LIN {X 0,Y 170.14,Z 485.3,A -85,B 0,C 180,E1 -24974.606,E2 -24974.606} C_VEL
LIN {X 0,Y 177.602,Z 482.481,A -85,B 0,C 180,E1 -24977.722,E2 -24977.722} C_VEL
LIN {X 0,Y 183.018,Z 480.013,A -85,B 0,C 180,E1 -24980.176,E2 -24980.176} C_VEL
LIN {X 0,Y 180.641,Z 479.716,A -85,B 0,C 180,E1 -24981.501,E2 -24981.501} C_VEL
LIN {X 0,Y 171.109,Z 479.234,A -85,B 0,C 180,E1 -24984.898,E2 -24984.898} C_VEL
LIN {X 0,Y 162.459,Z 477.57,A -85,B 0,C 180,E1 -24988.726,E2 -24988.726} C_VEL
LIN {X 0,Y 154.788,Z 474.682,A -85,B 0,C 180,E1 -24992.996,E2 -24992.996} C_VEL
LIN {X 0,Y 148.331,Z 470.573,A -85,B 0,C 180,E1 -24997.725,E2 -24997.725} C_VEL
LIN {X 0,Y 146.154,Z 468.596,A -85,B 0,C 180,E1 -24999.725,E2 -24999.725} C_VEL
LIN {X 0,Y 143.595,Z 466.459,A -85,B 0,C 180,E1 -25001.638,E2 -25001.638} C_VEL
LIN {X 0,Y 138.227,Z 462.461,A -85,B 0,C 180,E1 -25004.589,E2 -25004.589} C_VEL
LIN {X 0,Y 133.314,Z 457.777,A -85,B 0,C 180,E1 -25007.666,E2 -25007.666} C_VEL
LIN {X 0,Y 131.549,Z 454.712,A -85,B 0,C 180,E1 -25009.741,E2 -25009.741} C_VEL
LIN {X 0,Y 129.832,Z 446.19,A -85,B 0,C 180,E1 -25015.342,E2 -25015.342} C_VEL
LIN {X 0,Y 129.143,Z 437.874,A -85,B 0,C 180,E1 -25019.999,E2 -25019.999} C_VEL
LIN {X 0,Y 129.267,Z 426.337,A -85,B 0,C 180,E1 -25025.459,E2 -25025.459} C_VEL
LIN {X 0,Y 130.008,Z 415.476,A -85,B 0,C 180,E1 -25029.725,E2 -25029.725} C_VEL
LIN {X 0,Y 131.217,Z 402.421,A -85,B 0,C 180,E1 -25033.911,E2 -25033.911} C_VEL
LIN {X 0,Y 132.163,Z 391.334,A -85,B 0,C 180,E1 -25036.826,E2 -25036.826} C_VEL
LIN {X 0,Y 129.638,Z 379.334,A -85,B 0,C 180,E1 -25039.29,E2 -25039.29} C_VEL
LIN {X 0,Y 129.065,Z 379.401,A -85,B 0,C 180,E1 -25045.825,E2 -25045.825} C_VEL
LIN {X 0,Y 129.036,Z 379.412,A -85,B 0,C 180,E1 -25049.373,E2 -25049.373} C_VEL
LIN {X 0,Y 128.998,Z 379.412,A -85,B 0,C 180,E1 -25055.192,E2 -25055.192} C_VEL
LIN {X 0,Y 128.993,Z 379.414,A -85,B 0,C 180,E1 -25060.828,E2 -25060.828} C_VEL
LIN {X 0,Y 128.966,Z 379.42,A -85,B 0,C 180,E1 -25065.107,E2 -25065.107} C_VEL
LIN {X 0,Y 128.959,Z 379.418,A -85,B 0,C 180,E1 -25069.726,E2 -25069.726} C_VEL
LIN {X 0,Y 128.993,Z 379.418,A -85,B 0,C 180,E1 -25074.81,E2 -25074.81} C_VEL
LIN {X 0,Y 129.033,Z 379.406,A -85,B 0,C 180,E1 -25080.646,E2 -25080.646} C_VEL
LIN {X 0,Y 129.136,Z 379.395,A -85,B 0,C 180,E1 -25087.607,E2 -25087.607} C_VEL
LIN {X 0,Y 129.18,Z 379.392,A -85,B 0,C 180,E1 -25090.948,E2 -25090.948} C_VEL
LIN {X 0,Y 129.367,Z 379.364,A -85,B 0,C 180,E1 -25097.921,E2 -25097.921} C_VEL
LIN {X 0,Y 129.477,Z 379.357,A -85,B 0,C 180,E1 -25100.628,E2 -25100.628} C_VEL
LIN {X 0,Y 130.089,Z 379.282,A -85,B 0,C 180,E1 -25110,E2 -25110} C_VEL
LIN {X 0,Y 129.478,Z 379.357,A -85,B 0,C 180,E1 -25119.372,E2 -25119.372} C_VEL
LIN {X 0,Y 129.345,Z 379.366,A -85,B 0,C 180,E1 -25122.553,E2 -25122.553} C_VEL
LIN {X 0,Y 129.158,Z 379.395,A -85,B 0,C 180,E1 -25129.056,E2 -25129.056} C_VEL
LIN {X 0,Y 129.109,Z 379.398,A -85,B 0,C 180,E1 -25132.399,E2 -25132.399} C_VEL
LIN {X 0,Y 129.036,Z 379.406,A -85,B 0,C 180,E1 -25139.374,E2 -25139.374} C_VEL
LIN {X 0,Y 129.026,Z 379.414,A -85,B 0,C 180,E1 -25145.21,E2 -25145.21} C_VEL
LIN {X 0,Y 129.007,Z 379.413,A -85,B 0,C 180,E1 -25150.824,E2 -25150.824} C_VEL
LIN {X 0,Y 128.972,Z 379.417,A -85,B 0,C 180,E1 -25155.106,E2 -25155.106} C_VEL
LIN {X 0,Y 128.955,Z 379.421,A -85,B 0,C 180,E1 -25159.73,E2 -25159.73} C_VEL
LIN {X 0,Y 128.963,Z 379.416,A -85,B 0,C 180,E1 -25164.831,E2 -25164.831} C_VEL
LIN {X 0,Y 129.052,Z 379.41,A -85,B 0,C 180,E1 -25170.652,E2 -25170.652} C_VEL
LIN {X 0,Y 129.11,Z 379.402,A -85,B 0,C 180,E1 -25177.728,E2 -25177.728} C_VEL
LIN {X 0,Y 129.166,Z 379.392,A -85,B 0,C 180,E1 -25180.946,E2 -25180.946} C_VEL
LIN {X 0,Y 129.421,Z 379.363,A -85,B 0,C 180,E1 -25187.815,E2 -25187.815} C_VEL
LIN {X 0,Y 129.534,Z 379.344,A -85,B 0,C 180,E1 -25190.633,E2 -25190.633} C_VEL
LIN {X 0,Y 130.092,Z 379.274,A -85,B 0,C 180,E1 -25200,E2 -25200} C_VEL
LIN {X 0,Y 129.48,Z 379.351,A -85,B 0,C 180,E1 -25209.372,E2 -25209.372} C_VEL
LIN {X 0,Y 129.347,Z 379.373,A -85,B 0,C 180,E1 -25212.553,E2 -25212.553} C_VEL
LIN {X 0,Y 129.157,Z 379.394,A -85,B 0,C 180,E1 -25219.056,E2 -25219.056} C_VEL
LIN {X 0,Y 129.111,Z 379.402,A -85,B 0,C 180,E1 -25222.398,E2 -25222.398} C_VEL
LIN {X 0,Y 129.038,Z 379.411,A -85,B 0,C 180,E1 -25229.373,E2 -25229.373} C_VEL
LIN {X 0,Y 129.053,Z 379.404,A -85,B 0,C 180,E1 -25235.226,E2 -25235.226} C_VEL
LIN {X 0,Y 129.361,Z 379.369,A -85,B 0,C 180,E1 -25240.689,E2 -25240.689} C_VEL
LIN {X 0,Y 129.959,Z 379.326,A -85,B 0,C 180,E1 -25245.132,E2 -25245.132} C_VEL
LIN {X 0,Y 131.308,Z 383.898,A -85,B 0,C 180,E1 -25250.037,E2 -25250.037} C_VEL
LIN {X 0,Y 131.527,Z 385.753,A -85,B 0,C 180,E1 -25252.017,E2 -25252.017} C_VEL
LIN {X 0,Y 130.174,Z 390.538,A -85,B 0,C 180,E1 -25257.323,E2 -25257.323} C_VEL
LIN {X 0,Y 128.998,Z 398.088,A -85,B 0,C 180,E1 -25265.989,E2 -25265.989} C_VEL
LIN {X 0,Y 128.362,Z 411.728,A -85,B 0,C 180,E1 -25268.252,E2 -25268.252} C_VEL
LIN {X 0,Y 128.633,Z 424.364,A -85,B 0,C 180,E1 -25270.863,E2 -25270.863} C_VEL
LIN {X 0,Y 129.819,Z 437.824,A -85,B 0,C 180,E1 -25274.295,E2 -25274.295} C_VEL
LIN {X 0,Y 131.612,Z 449.97,A -85,B 0,C 180,E1 -25278.058,E2 -25278.058} C_VEL
LIN {X 0,Y 132.698,Z 455.665,A -85,B 0,C 180,E1 -25280.088,E2 -25280.088} C_VEL
LIN {X 0,Y 133.201,Z 464.15,A -85,B 0,C 180,E1 -25283.942,E2 -25283.942} C_VEL
LIN {X 0,Y 133.939,Z 470.787,A -85,B 0,C 180,E1 -25287.567,E2 -25287.567} C_VEL
LIN {X 0,Y 135.046,Z 476.747,A -85,B 0,C 180,E1 -25291.491,E2 -25291.491} C_VEL
LIN {X 0,Y 134.77,Z 478.314,A -85,B 0,C 180,E1 -25292.989,E2 -25292.989} C_VEL
LIN {X 0,Y 132.305,Z 482.493,A -85,B 0,C 180,E1 -25299.17,E2 -25299.17} C_VEL
LIN {X 0,Y 131.65,Z 485.641,A -85,B 0,C 180,E1 -25306.071,E2 -25306.071} C_VEL
LIN {X 0,Y 132.923,Z 487.379,A -85,B 0,C 180,E1 -25311.722,E2 -25311.722} C_VEL
LIN {X 0,Y 136.259,Z 488.459,A -85,B 0,C 180,E1 -25317.659,E2 -25317.659} C_VEL
LIN {X 0,Y 141.551,Z 488.732,A -85,B 0,C 180,E1 -25323.103,E2 -25323.103} C_VEL
LIN {X 0,Y 148.341,Z 488.17,A -85,B 0,C 180,E1 -25328.018,E2 -25328.018} C_VEL
LIN {X 0,Y 156.192,Z 486.763,A -85,B 0,C 180,E1 -25332.45,E2 -25332.45} C_VEL
LIN {X 0,Y 165.142,Z 484.583,A -85,B 0,C 180,E1 -25336.342,E2 -25336.342} C_VEL
LIN {X 0,Y 172.211,Z 482.323,A -85,B 0,C 180,E1 -25339.234,E2 -25339.234} C_VEL
LIN {X 0,Y 174.086,Z 481.574,A -85,B 0,C 180,E1 -25340.09,E2 -25340.09} C_VEL
LIN {X 0,Y 169.266,Z 480.977,A -85,B 0,C 180,E1 -25342.082,E2 -25342.082} C_VEL
LIN {X 0,Y 160.81,Z 479.531,A -85,B 0,C 180,E1 -25345.378,E2 -25345.378} C_VEL
LIN {X 0,Y 152.361,Z 476.82,A -85,B 0,C 180,E1 -25349.509,E2 -25349.509} C_VEL
LIN {X 0,Y 144.959,Z 472.908,A -85,B 0,C 180,E1 -25354.129,E2 -25354.129} C_VEL
LIN {X 0,Y 138.954,Z 467.741,A -85,B 0,C 180,E1 -25359.265,E2 -25359.265} C_VEL
LIN {X 0,Y 134.271,Z 461.25,A -85,B 0,C 180,E1 -25364.828,E2 -25364.828} C_VEL
LIN {X 0,Y 131.549,Z 454.712,A -85,B 0,C 180,E1 -25369.741,E2 -25369.741} C_VEL
LIN {X 0,Y 130.004,Z 451.514,A -85,B 0,C 180,E1 -25371.813,E2 -25371.813} C_VEL
LIN {X 0,Y 126.277,Z 445.65,A -85,B 0,C 180,E1 -25374.992,E2 -25374.992} C_VEL
LIN {X 0,Y 122.987,Z 439.301,A -85,B 0,C 180,E1 -25378.18,E2 -25378.18} C_VEL
LIN {X 0,Y 122.189,Z 435.308,A -85,B 0,C 180,E1 -25380.201,E2 -25380.201} C_VEL
LIN {X 0,Y 122.392,Z 423.535,A -85,B 0,C 180,E1 -25385.767,E2 -25385.767} C_VEL
LIN {X 0,Y 123.115,Z 413.168,A -85,B 0,C 180,E1 -25389.86,E2 -25389.86} C_VEL
LIN {X 0,Y 124.272,Z 400.77,A -85,B 0,C 180,E1 -25393.907,E2 -25393.907} C_VEL
LIN {X 0,Y 125.093,Z 391.958,A -85,B 0,C 180,E1 -25396.314,E2 -25396.314} C_VEL
LIN {X 0,Y 122.644,Z 380.202,A -85,B 0,C 180,E1 -25398.911,E2 -25398.911} C_VEL
LIN {X 0,Y 121.974,Z 380.289,A -85,B 0,C 180,E1 -25407.448,E2 -25407.448} C_VEL
LIN {X 0,Y 121.913,Z 380.298,A -85,B 0,C 180,E1 -25411.253,E2 -25411.253} C_VEL
LIN {X 0,Y 121.922,Z 380.294,A -85,B 0,C 180,E1 -25416.195,E2 -25416.195} C_VEL
LIN {X 0,Y 121.92,Z 380.293,A -85,B 0,C 180,E1 -25421.464,E2 -25421.464} C_VEL
LIN {X 0,Y 121.891,Z 380.301,A -85,B 0,C 180,E1 -25428.551,E2 -25428.551} C_VEL
LIN {X 0,Y 121.946,Z 380.296,A -85,B 0,C 180,E1 -25434.808,E2 -25434.808} C_VEL
LIN {X 0,Y 121.942,Z 380.289,A -85,B 0,C 180,E1 -25439.826,E2 -25439.826} C_VEL
LIN {X 0,Y 122.068,Z 380.275,A -85,B 0,C 180,E1 -25447.1,E2 -25447.1} C_VEL
LIN {X 0,Y 122.122,Z 380.272,A -85,B 0,C 180,E1 -25453.277,E2 -25453.277} C_VEL
LIN {X 0,Y 122.318,Z 380.241,A -85,B 0,C 180,E1 -25457.623,E2 -25457.623} C_VEL
LIN {X 0,Y 122.426,Z 380.233,A -85,B 0,C 180,E1 -25463.407,E2 -25463.407} C_VEL
LIN {X 0,Y 123.043,Z 380.159,A -85,B 0,C 180,E1 -25470,E2 -25470} C_VEL
LIN {X 0,Y 122.427,Z 380.233,A -85,B 0,C 180,E1 -25476.593,E2 -25476.593} C_VEL
LIN {X 0,Y 122.318,Z 380.241,A -85,B 0,C 180,E1 -25482.377,E2 -25482.377} C_VEL
LIN {X 0,Y 122.112,Z 380.273,A -85,B 0,C 180,E1 -25486.725,E2 -25486.725} C_VEL
LIN {X 0,Y 122.024,Z 380.281,A -85,B 0,C 180,E1 -25492.852,E2 -25492.852} C_VEL
LIN {X 0,Y 121.95,Z 380.293,A -85,B 0,C 180,E1 -25497.455,E2 -25497.455} C_VEL
LIN {X 0,Y 121.913,Z 380.294,A -85,B 0,C 180,E1 -25501.254,E2 -25501.254} C_VEL
LIN {X 0,Y 121.939,Z 380.293,A -85,B 0,C 180,E1 -25506.207,E2 -25506.207} C_VEL
LIN {X 0,Y 121.931,Z 380.296,A -85,B 0,C 180,E1 -25511.47,E2 -25511.47} C_VEL
LIN {X 0,Y 121.892,Z 380.297,A -85,B 0,C 180,E1 -25518.552,E2 -25518.552} C_VEL
LIN {X 0,Y 121.915,Z 380.293,A -85,B 0,C 180,E1 -25524.798,E2 -25524.798} C_VEL
LIN {X 0,Y 121.941,Z 380.295,A -85,B 0,C 180,E1 -25529.829,E2 -25529.829} C_VEL
LIN {X 0,Y 121.986,Z 380.287,A -85,B 0,C 180,E1 -25536.216,E2 -25536.216} C_VEL
LIN {X 0,Y 122.054,Z 380.28,A -85,B 0,C 180,E1 -25539.789,E2 -25539.789} C_VEL
LIN {X 0,Y 122.289,Z 380.253,A -85,B 0,C 180,E1 -25546.71,E2 -25546.71} C_VEL
LIN {X 0,Y 122.46,Z 380.228,A -85,B 0,C 180,E1 -25550.086,E2 -25550.086} C_VEL
LIN {X 0,Y 122.614,Z 380.211,A -85,B 0,C 180,E1 -25556.715,E2 -25556.715} C_VEL
LIN {X 0,Y 123.045,Z 380.151,A -85,B 0,C 180,E1 -25560.001,E2 -25560.001} C_VEL
LIN {X 0,Y 122.428,Z 380.232,A -85,B 0,C 180,E1 -25566.593,E2 -25566.593} C_VEL
LIN {X 0,Y 122.32,Z 380.249,A -85,B 0,C 180,E1 -25572.377,E2 -25572.377} C_VEL
LIN {X 0,Y 122.111,Z 380.267,A -85,B 0,C 180,E1 -25576.725,E2 -25576.725} C_VEL
LIN {X 0,Y 122.026,Z 380.283,A -85,B 0,C 180,E1 -25582.851,E2 -25582.851} C_VEL
LIN {X 0,Y 121.952,Z 380.29,A -85,B 0,C 180,E1 -25587.454,E2 -25587.454} C_VEL
LIN {X 0,Y 121.917,Z 380.298,A -85,B 0,C 180,E1 -25591.253,E2 -25591.253} C_VEL
LIN {X 0,Y 122.037,Z 380.282,A -85,B 0,C 180,E1 -25596.268,E2 -25596.268} C_VEL
LIN {X 0,Y 122.898,Z 380.18,A -85,B 0,C 180,E1 -25605.125,E2 -25605.125} C_VEL
LIN {X 0,Y 123.1,Z 380.269,A -85,B 0,C 180,E1 -25606.284,E2 -25606.284} C_VEL
LIN {X 0,Y 124.019,Z 383.15,A -85,B 0,C 180,E1 -25609.562,E2 -25609.562} C_VEL
LIN {X 0,Y 124.38,Z 385.558,A -85,B 0,C 180,E1 -25612.286,E2 -25612.286} C_VEL
LIN {X 0,Y 123.156,Z 389.67,A -85,B 0,C 180,E1 -25617.171,E2 -25617.171} C_VEL
LIN {X 0,Y 122.005,Z 397.074,A -85,B 0,C 180,E1 -25626.298,E2 -25626.298} C_VEL
LIN {X 0,Y 121.409,Z 409.093,A -85,B 0,C 180,E1 -25628.377,E2 -25628.377} C_VEL
LIN {X 0,Y 121.725,Z 423.36,A -85,B 0,C 180,E1 -25631.485,E2 -25631.485} C_VEL
LIN {X 0,Y 123.055,Z 437.085,A -85,B 0,C 180,E1 -25635.204,E2 -25635.204} C_VEL
LIN {X 0,Y 124.946,Z 448.82,A -85,B 0,C 180,E1 -25639.056,E2 -25639.056} C_VEL
LIN {X 0,Y 126.146,Z 454.516,A -85,B 0,C 180,E1 -25641.187,E2 -25641.187} C_VEL
LIN {X 0,Y 126.68,Z 461.745,A -85,B 0,C 180,E1 -25644.633,E2 -25644.633} C_VEL
LIN {X 0,Y 127.616,Z 468.962,A -85,B 0,C 180,E1 -25648.725,E2 -25648.725} C_VEL
LIN {X 0,Y 128.474,Z 473.274,A -85,B 0,C 180,E1 -25651.567,E2 -25651.567} C_VEL
LIN {X 0,Y 128.453,Z 475.044,A -85,B 0,C 180,E1 -25653.136,E2 -25653.136} C_VEL
LIN {X 0,Y 125.905,Z 479.435,A -85,B 0,C 180,E1 -25659.64,E2 -25659.64} C_VEL
LIN {X 0,Y 125.383,Z 483.15,A -85,B 0,C 180,E1 -25667.655,E2 -25667.655} C_VEL
LIN {X 0,Y 128.252,Z 485.578,A -85,B 0,C 180,E1 -25676.001,E2 -25676.001} C_VEL
LIN {X 0,Y 133.627,Z 486.621,A -85,B 0,C 180,E1 -25682.699,E2 -25682.699} C_VEL
LIN {X 0,Y 142.919,Z 486.504,A -85,B 0,C 180,E1 -25689.738,E2 -25689.738} C_VEL
LIN {X 0,Y 151.093,Z 485.444,A -85,B 0,C 180,E1 -25694.244,E2 -25694.244} C_VEL
LIN {X 0,Y 160.329,Z 483.66,A -85,B 0,C 180,E1 -25698.176,E2 -25698.176} C_VEL
LIN {X 0,Y 165.008,Z 482.426,A -85,B 0,C 180,E1 -25700.054,E2 -25700.054} C_VEL
LIN {X 0,Y 159.837,Z 481.469,A -85,B 0,C 180,E1 -25702.006,E2 -25702.006} C_VEL
LIN {X 0,Y 150.542,Z 478.882,A -85,B 0,C 180,E1 -25705.929,E2 -25705.929} C_VEL
LIN {X 0,Y 142.294,Z 475.138,A -85,B 0,C 180,E1 -25710.402,E2 -25710.402} C_VEL
LIN {X 0,Y 135.297,Z 470.197,A -85,B 0,C 180,E1 -25715.445,E2 -25715.445} C_VEL
LIN {X 0,Y 129.736,Z 463.945,A -85,B 0,C 180,E1 -25721.032,E2 -25721.032} C_VEL
LIN {X 0,Y 125.658,Z 456.29,A -85,B 0,C 180,E1 -25727.072,E2 -25727.072} C_VEL
LIN {X 0,Y 123.222,Z 447.02,A -85,B 0,C 180,E1 -25733.449,E2 -25733.449} C_VEL
LIN {X 0,Y 122.396,Z 438.754,A -85,B 0,C 180,E1 -25738.354,E2 -25738.354} C_VEL
LIN {X 0,Y 122.189,Z 435.308,A -85,B 0,C 180,E1 -25740.201,E2 -25740.201} C_VEL
LIN {X 0,Y 121.505,Z 431.227,A -85,B 0,C 180,E1 -25742.158,E2 -25742.158} C_VEL
LIN {X 0,Y 118.944,Z 423.968,A -85,B 0,C 180,E1 -25745.092,E2 -25745.092} C_VEL
LIN {X 0,Y 116.555,Z 416.203,A -85,B 0,C 180,E1 -25747.953,E2 -25747.953} C_VEL
LIN {X 0,Y 116.228,Z 411.378,A -85,B 0,C 180,E1 -25749.71,E2 -25749.71} C_VEL
LIN {X 0,Y 117.336,Z 399.012,A -85,B 0,C 180,E1 -25753.862,E2 -25753.862} C_VEL
LIN {X 0,Y 117.981,Z 391.979,A -85,B 0,C 180,E1 -25755.837,E2 -25755.837} C_VEL
LIN {X 0,Y 115.703,Z 381.064,A -85,B 0,C 180,E1 -25758.366,E2 -25758.366} C_VEL
LIN {X 0,Y 114.949,Z 381.159,A -85,B 0,C 180,E1 -25765.339,E2 -25765.339} C_VEL
LIN {X 0,Y 114.871,Z 381.176,A -85,B 0,C 180,E1 -25771.069,E2 -25771.069} C_VEL
LIN {X 0,Y 114.822,Z 381.182,A -85,B 0,C 180,E1 -25777.739,E2 -25777.739} C_VEL
LIN {X 0,Y 114.832,Z 381.174,A -85,B 0,C 180,E1 -25782.741,E2 -25782.741} C_VEL
LIN {X 0,Y 114.819,Z 381.182,A -85,B 0,C 180,E1 -25787.677,E2 -25787.677} C_VEL
LIN {X 0,Y 114.812,Z 381.178,A -85,B 0,C 180,E1 -25792.727,E2 -25792.727} C_VEL
LIN {X 0,Y 114.869,Z 381.17,A -85,B 0,C 180,E1 -25798.931,E2 -25798.931} C_VEL
LIN {X 0,Y 114.966,Z 381.161,A -85,B 0,C 180,E1 -25806.485,E2 -25806.485} C_VEL
LIN {X 0,Y 115.027,Z 381.157,A -85,B 0,C 180,E1 -25812.212,E2 -25812.212} C_VEL
LIN {X 0,Y 115.252,Z 381.121,A -85,B 0,C 180,E1 -25817.333,E2 -25817.333} C_VEL
LIN {X 0,Y 115.367,Z 381.113,A -85,B 0,C 180,E1 -25823.002,E2 -25823.002} C_VEL
LIN {X 0,Y 115.994,Z 381.037,A -85,B 0,C 180,E1 -25830,E2 -25830} C_VEL
LIN {X 0,Y 115.367,Z 381.113,A -85,B 0,C 180,E1 -25836.998,E2 -25836.998} C_VEL
LIN {X 0,Y 115.252,Z 381.121,A -85,B 0,C 180,E1 -25842.667,E2 -25842.667} C_VEL
LIN {X 0,Y 115.014,Z 381.159,A -85,B 0,C 180,E1 -25847.79,E2 -25847.79} C_VEL
LIN {X 0,Y 114.947,Z 381.164,A -85,B 0,C 180,E1 -25853.493,E2 -25853.493} C_VEL
LIN {X 0,Y 114.87,Z 381.17,A -85,B 0,C 180,E1 -25861.069,E2 -25861.069} C_VEL
LIN {X 0,Y 114.849,Z 381.172,A -85,B 0,C 180,E1 -25867.73,E2 -25867.73} C_VEL
LIN {X 0,Y 114.842,Z 381.18,A -85,B 0,C 180,E1 -25872.747,E2 -25872.747} C_VEL
LIN {X 0,Y 114.821,Z 381.176,A -85,B 0,C 180,E1 -25877.679,E2 -25877.679} C_VEL
LIN {X 0,Y 114.795,Z 381.186,A -85,B 0,C 180,E1 -25882.74,E2 -25882.74} C_VEL
LIN {X 0,Y 114.864,Z 381.177,A -85,B 0,C 180,E1 -25888.938,E2 -25888.938} C_VEL
LIN {X 0,Y 114.949,Z 381.164,A -85,B 0,C 180,E1 -25896.508,E2 -25896.508} C_VEL
LIN {X 0,Y 115.023,Z 381.151,A -85,B 0,C 180,E1 -25902.212,E2 -25902.212} C_VEL
LIN {X 0,Y 115.289,Z 381.124,A -85,B 0,C 180,E1 -25907.258,E2 -25907.258} C_VEL
LIN {X 0,Y 115.396,Z 381.108,A -85,B 0,C 180,E1 -25909.473,E2 -25909.473} C_VEL
LIN {X 0,Y 115.541,Z 381.093,A -85,B 0,C 180,E1 -25916.513,E2 -25916.513} C_VEL
LIN {X 0,Y 115.997,Z 381.029,A -85,B 0,C 180,E1 -25920.001,E2 -25920.001} C_VEL
LIN {X 0,Y 115.369,Z 381.11,A -85,B 0,C 180,E1 -25926.999,E2 -25926.999} C_VEL
LIN {X 0,Y 115.255,Z 381.129,A -85,B 0,C 180,E1 -25932.667,E2 -25932.667} C_VEL
LIN {X 0,Y 115.014,Z 381.151,A -85,B 0,C 180,E1 -25937.791,E2 -25937.791} C_VEL
LIN {X 0,Y 114.95,Z 381.165,A -85,B 0,C 180,E1 -25943.493,E2 -25943.493} C_VEL
LIN {X 0,Y 114.874,Z 381.175,A -85,B 0,C 180,E1 -25951.07,E2 -25951.07} C_VEL
LIN {X 0,Y 115.033,Z 381.155,A -85,B 0,C 180,E1 -25957.659,E2 -25957.659} C_VEL
LIN {X 0,Y 116.078,Z 381.03,A -85,B 0,C 180,E1 -25966.599,E2 -25966.599} C_VEL
LIN {X 0,Y 116.265,Z 381.092,A -85,B 0,C 180,E1 -25967.535,E2 -25967.535} C_VEL
LIN {X 0,Y 117.185,Z 384.161,A -85,B 0,C 180,E1 -25971.23,E2 -25971.23} C_VEL
LIN {X 0,Y 117.073,Z 385.702,A -85,B 0,C 180,E1 -25973.107,E2 -25973.107} C_VEL
LIN {X 0,Y 115.477,Z 391.71,A -85,B 0,C 180,E1 -25980.863,E2 -25980.863} C_VEL
LIN {X 0,Y 115.018,Z 396.094,A -85,B 0,C 180,E1 -25986.675,E2 -25986.675} C_VEL
LIN {X 0,Y 114.46,Z 407.836,A -85,B 0,C 180,E1 -25988.854,E2 -25988.854} C_VEL
LIN {X 0,Y 114.832,Z 422.144,A -85,B 0,C 180,E1 -25992.18,E2 -25992.18} C_VEL
LIN {X 0,Y 116.245,Z 435.48,A -85,B 0,C 180,E1 -25996.005,E2 -25996.005} C_VEL
LIN {X 0,Y 118.355,Z 447.553,A -85,B 0,C 180,E1 -26000.17,E2 -26000.17} C_VEL
LIN {X 0,Y 119.663,Z 453.235,A -85,B 0,C 180,E1 -26002.406,E2 -26002.406} C_VEL
LIN {X 0,Y 120.475,Z 461.551,A -85,B 0,C 180,E1 -26006.655,E2 -26006.655} C_VEL
LIN {X 0,Y 121.894,Z 469.512,A -85,B 0,C 180,E1 -26011.652,E2 -26011.652} C_VEL
LIN {X 0,Y 122.132,Z 471.597,A -85,B 0,C 180,E1 -26013.299,E2 -26013.299} C_VEL
LIN {X 0,Y 120.461,Z 474.552,A -85,B 0,C 180,E1 -26017.326,E2 -26017.326} C_VEL
LIN {X 0,Y 119.036,Z 478.093,A -85,B 0,C 180,E1 -26023.66,E2 -26023.66} C_VEL
LIN {X 0,Y 119.56,Z 480.975,A -85,B 0,C 180,E1 -26030.652,E2 -26030.652} C_VEL
LIN {X 0,Y 122.273,Z 482.983,A -85,B 0,C 180,E1 -26037.376,E2 -26037.376} C_VEL
LIN {X 0,Y 128.681,Z 484.429,A -85,B 0,C 180,E1 -26044.99,E2 -26044.99} C_VEL
LIN {X 0,Y 137.686,Z 484.661,A -85,B 0,C 180,E1 -26051.573,E2 -26051.573} C_VEL
LIN {X 0,Y 146.172,Z 483.928,A -85,B 0,C 180,E1 -26056.154,E2 -26056.154} C_VEL
LIN {X 0,Y 150.86,Z 483.324,A -85,B 0,C 180,E1 -26058.192,E2 -26058.192} C_VEL
LIN {X 0,Y 154.336,Z 482.295,A -85,B 0,C 180,E1 -26060.393,E2 -26060.393} C_VEL
LIN {X 0,Y 144.732,Z 479.243,A -85,B 0,C 180,E1 -26064.358,E2 -26064.358} C_VEL
LIN {X 0,Y 136.178,Z 475.05,A -85,B 0,C 180,E1 -26068.929,E2 -26068.929} C_VEL
LIN {X 0,Y 128.883,Z 469.671,A -85,B 0,C 180,E1 -26074.135,E2 -26074.135} C_VEL
LIN {X 0,Y 123.086,Z 463.014,A -85,B 0,C 180,E1 -26079.965,E2 -26079.965} C_VEL
LIN {X 0,Y 118.441,Z 453.782,A -85,B 0,C 180,E1 -26087.143,E2 -26087.143} C_VEL
LIN {X 0,Y 116.367,Z 445.166,A -85,B 0,C 180,E1 -26093.062,E2 -26093.062} C_VEL
LIN {X 0,Y 115.471,Z 436.462,A -85,B 0,C 180,E1 -26098.256,E2 -26098.256} C_VEL
LIN {X 0,Y 115.407,Z 424.357,A -85,B 0,C 180,E1 -26104.365,E2 -26104.365} C_VEL
LIN {X 0,Y 116.038,Z 414.064,A -85,B 0,C 180,E1 -26108.708,E2 -26108.708} C_VEL
LIN {X 0,Y 116.228,Z 411.378,A -85,B 0,C 180,E1 -26109.71,E2 -26109.71} C_VEL
LIN {X 0,Y 115.939,Z 406.526,A -85,B 0,C 180,E1 -26111.367,E2 -26111.367} C_VEL
LIN {X 0,Y 114.723,Z 401.509,A -85,B 0,C 180,E1 -26112.857,E2 -26112.857} C_VEL
LIN {X 0,Y 111.131,Z 391.201,A -85,B 0,C 180,E1 -26115.515,E2 -26115.515} C_VEL
LIN {X 0,Y 109.189,Z 384.008,A -85,B 0,C 180,E1 -26117.164,E2 -26117.164} C_VEL
LIN {X 0,Y 108.789,Z 381.923,A -85,B 0,C 180,E1 -26117.674,E2 -26117.674} C_VEL
LIN {X 0,Y 107.83,Z 382.048,A -85,B 0,C 180,E1 -26127.144,E2 -26127.144} C_VEL
LIN {X 0,Y 107.797,Z 382.055,A -85,B 0,C 180,E1 -26132.053,E2 -26132.053} C_VEL
LIN {X 0,Y 107.729,Z 382.066,A -85,B 0,C 180,E1 -26138.477,E2 -26138.477} C_VEL
LIN {X 0,Y 107.705,Z 382.068,A -85,B 0,C 180,E1 -26145.87,E2 -26145.87} C_VEL
LIN {X 0,Y 107.71,Z 382.06,A -85,B 0,C 180,E1 -26151.534,E2 -26151.534} C_VEL
LIN {X 0,Y 107.807,Z 382.051,A -85,B 0,C 180,E1 -26158.566,E2 -26158.566} C_VEL
LIN {X 0,Y 107.931,Z 382.036,A -85,B 0,C 180,E1 -26167.002,E2 -26167.002} C_VEL
LIN {X 0,Y 108.036,Z 382.025,A -85,B 0,C 180,E1 -26174.918,E2 -26174.918} C_VEL
LIN {X 0,Y 108.254,Z 381.997,A -85,B 0,C 180,E1 -26178.769,E2 -26178.769} C_VEL
LIN {X 0,Y 108.448,Z 381.97,A -85,B 0,C 180,E1 -26186.285,E2 -26186.285} C_VEL
LIN {X 0,Y 108.944,Z 381.915,A -85,B 0,C 180,E1 -26190,E2 -26190} C_VEL
LIN {X 0,Y 108.305,Z 381.993,A -85,B 0,C 180,E1 -26197.457,E2 -26197.457} C_VEL
LIN {X 0,Y 108.173,Z 382.002,A -85,B 0,C 180,E1 -26202.957,E2 -26202.957} C_VEL
LIN {X 0,Y 107.906,Z 382.042,A -85,B 0,C 180,E1 -26209.006,E2 -26209.006} C_VEL
LIN {X 0,Y 107.858,Z 382.049,A -85,B 0,C 180,E1 -26214.185,E2 -26214.185} C_VEL
LIN {X 0,Y 107.8,Z 382.055,A -85,B 0,C 180,E1 -26222.057,E2 -26222.057} C_VEL
LIN {X 0,Y 107.751,Z 382.055,A -85,B 0,C 180,E1 -26228.493,E2 -26228.493} C_VEL
LIN {X 0,Y 107.709,Z 382.063,A -85,B 0,C 180,E1 -26235.87,E2 -26235.87} C_VEL
LIN {X 0,Y 107.699,Z 382.07,A -85,B 0,C 180,E1 -26241.544,E2 -26241.544} C_VEL
LIN {X 0,Y 107.799,Z 382.055,A -85,B 0,C 180,E1 -26248.564,E2 -26248.564} C_VEL
LIN {X 0,Y 107.913,Z 382.042,A -85,B 0,C 180,E1 -26256.999,E2 -26256.999} C_VEL
LIN {X 0,Y 108.049,Z 382.023,A -85,B 0,C 180,E1 -26264.92,E2 -26264.92} C_VEL
LIN {X 0,Y 108.309,Z 381.992,A -85,B 0,C 180,E1 -26268.775,E2 -26268.775} C_VEL
LIN {X 0,Y 108.466,Z 381.975,A -85,B 0,C 180,E1 -26276.286,E2 -26276.286} C_VEL
LIN {X 0,Y 108.946,Z 381.907,A -85,B 0,C 180,E1 -26280.001,E2 -26280.001} C_VEL
LIN {X 0,Y 108.307,Z 381.989,A -85,B 0,C 180,E1 -26287.457,E2 -26287.457} C_VEL
LIN {X 0,Y 108.175,Z 382.01,A -85,B 0,C 180,E1 -26292.956,E2 -26292.956} C_VEL
LIN {X 0,Y 107.907,Z 382.041,A -85,B 0,C 180,E1 -26299.006,E2 -26299.006} C_VEL
LIN {X 0,Y 107.86,Z 382.045,A -85,B 0,C 180,E1 -26304.185,E2 -26304.185} C_VEL
LIN {X 0,Y 107.808,Z 382.053,A -85,B 0,C 180,E1 -26312.061,E2 -26312.061} C_VEL
LIN {X 0,Y 108.147,Z 382.012,A -85,B 0,C 180,E1 -26320.532,E2 -26320.532} C_VEL
LIN {X 0,Y 109.512,Z 381.873,A -85,B 0,C 180,E1 -26328.944,E2 -26328.944} C_VEL
LIN {X 0,Y 109.851,Z 382.874,A -85,B 0,C 180,E1 -26330.224,E2 -26330.224} C_VEL
LIN {X 0,Y 110.024,Z 384.729,A -85,B 0,C 180,E1 -26332.639,E2 -26332.639} C_VEL
LIN {X 0,Y 108.724,Z 389.222,A -85,B 0,C 180,E1 -26338.86,E2 -26338.86} C_VEL
LIN {X 0,Y 108.067,Z 395.013,A -85,B 0,C 180,E1 -26347.159,E2 -26347.159} C_VEL
LIN {X 0,Y 107.551,Z 407.596,A -85,B 0,C 180,E1 -26349.687,E2 -26349.687} C_VEL
LIN {X 0,Y 107.99,Z 420.747,A -85,B 0,C 180,E1 -26352.97,E2 -26352.97} C_VEL
LIN {X 0,Y 109.543,Z 434.095,A -85,B 0,C 180,E1 -26357.027,E2 -26357.027} C_VEL
LIN {X 0,Y 111.83,Z 446.154,A -85,B 0,C 180,E1 -26361.416,E2 -26361.416} C_VEL
LIN {X 0,Y 113.366,Z 452.763,A -85,B 0,C 180,E1 -26364.214,E2 -26364.214} C_VEL
LIN {X 0,Y 114.508,Z 461.538,A -85,B 0,C 180,E1 -26369.121,E2 -26369.121} C_VEL
LIN {X 0,Y 115.894,Z 467.951,A -85,B 0,C 180,E1 -26373.476,E2 -26373.476} C_VEL
LIN {X 0,Y 114.516,Z 470.672,A -85,B 0,C 180,E1 -26377.05,E2 -26377.05} C_VEL
LIN {X 0,Y 112.839,Z 474.848,A -85,B 0,C 180,E1 -26384.426,E2 -26384.426} C_VEL
LIN {X 0,Y 113.477,Z 477.975,A -85,B 0,C 180,E1 -26391.814,E2 -26391.814} C_VEL
LIN {X 0,Y 116.446,Z 480.221,A -85,B 0,C 180,E1 -26398.871,E2 -26398.871} C_VEL
LIN {X 0,Y 121.651,Z 481.759,A -85,B 0,C 180,E1 -26405.29,E2 -26405.29} C_VEL
LIN {X 0,Y 128.602,Z 482.537,A -85,B 0,C 180,E1 -26410.98,E2 -26410.98} C_VEL
LIN {X 0,Y 141.463,Z 482.217,A -85,B 0,C 180,E1 -26418.178,E2 -26418.178} C_VEL
LIN {X 0,Y 144.373,Z 481.986,A -85,B 0,C 180,E1 -26419.436,E2 -26419.436} C_VEL
LIN {X 0,Y 143.839,Z 481.289,A -85,B 0,C 180,E1 -26420.566,E2 -26420.566} C_VEL
LIN {X 0,Y 134.455,Z 477.217,A -85,B 0,C 180,E1 -26424.902,E2 -26424.902} C_VEL
LIN {X 0,Y 126.146,Z 471.985,A -85,B 0,C 180,E1 -26429.905,E2 -26429.905} C_VEL
LIN {X 0,Y 119.372,Z 465.547,A -85,B 0,C 180,E1 -26435.661,E2 -26435.661} C_VEL
LIN {X 0,Y 114.101,Z 457.746,A -85,B 0,C 180,E1 -26442.062,E2 -26442.062} C_VEL
LIN {X 0,Y 110.576,Z 448.356,A -85,B 0,C 180,E1 -26449.007,E2 -26449.007} C_VEL
LIN {X 0,Y 109.025,Z 438.639,A -85,B 0,C 180,E1 -26455.378,E2 -26455.378} C_VEL
LIN {X 0,Y 108.438,Z 426.844,A -85,B 0,C 180,E1 -26461.856,E2 -26461.856} C_VEL
LIN {X 0,Y 109.015,Z 414.776,A -85,B 0,C 180,E1 -26467.408,E2 -26467.408} C_VEL
LIN {X 0,Y 110.104,Z 401.216,A -85,B 0,C 180,E1 -26472.44,E2 -26472.44} C_VEL
LIN {X 0,Y 110.894,Z 391.893,A -85,B 0,C 180,E1 -26475.275,E2 -26475.275} C_VEL
LIN {X 0,Y 109.189,Z 384.008,A -85,B 0,C 180,E1 -26477.164,E2 -26477.164} C_VEL
LIN {X 0,Y 108.623,Z 382.755,A -85,B 0,C 180,E1 -26477.814,E2 -26477.814} C_VEL
LIN {X 0,Y 107.486,Z 382.185,A -85,B 0,C 180,E1 -26479.145,E2 -26479.145} C_VEL
LIN {X 0,Y 104.036,Z 382.522,A -85,B 0,C 180,E1 -26483.899,E2 -26483.899} C_VEL
LIN {X 0,Y 101.665,Z 383.072,A -85,B 0,C 180,E1 -26488.763,E2 -26488.763} C_VEL
LIN {X 0,Y 100.686,Z 382.935,A -85,B 0,C 180,E1 -26493.879,E2 -26493.879} C_VEL
LIN {X 0,Y 100.678,Z 382.943,A -85,B 0,C 180,E1 -26499.836,E2 -26499.836} C_VEL
LIN {X 0,Y 100.676,Z 382.943,A -85,B 0,C 180,E1 -26505.726,E2 -26505.726} C_VEL
LIN {X 0,Y 100.649,Z 382.94,A -85,B 0,C 180,E1 -26511.065,E2 -26511.065} C_VEL
LIN {X 0,Y 100.7,Z 382.94,A -85,B 0,C 180,E1 -26516.876,E2 -26516.876} C_VEL
LIN {X 0,Y 100.786,Z 382.93,A -85,B 0,C 180,E1 -26525.267,E2 -26525.267} C_VEL
LIN {X 0,Y 100.835,Z 382.919,A -85,B 0,C 180,E1 -26529.605,E2 -26529.605} C_VEL
LIN {X 0,Y 101.102,Z 382.883,A -85,B 0,C 180,E1 -26536.702,E2 -26536.702} C_VEL
LIN {X 0,Y 101.243,Z 382.874,A -85,B 0,C 180,E1 -26542.02,E2 -26542.02} C_VEL
LIN {X 0,Y 101.867,Z 382.797,A -85,B 0,C 180,E1 -26550,E2 -26550} C_VEL
LIN {X 0,Y 101.244,Z 382.874,A -85,B 0,C 180,E1 -26557.981,E2 -26557.981} C_VEL
LIN {X 0,Y 101.102,Z 382.883,A -85,B 0,C 180,E1 -26563.299,E2 -26563.299} C_VEL
LIN {X 0,Y 100.817,Z 382.921,A -85,B 0,C 180,E1 -26570.399,E2 -26570.399} C_VEL
LIN {X 0,Y 100.774,Z 382.931,A -85,B 0,C 180,E1 -26574.959,E2 -26574.959} C_VEL
LIN {X 0,Y 100.708,Z 382.939,A -85,B 0,C 180,E1 -26583.131,E2 -26583.131} C_VEL
LIN {X 0,Y 100.694,Z 382.937,A -85,B 0,C 180,E1 -26589.849,E2 -26589.849} C_VEL
LIN {X 0,Y 100.68,Z 382.939,A -85,B 0,C 180,E1 -26595.73,E2 -26595.73} C_VEL
LIN {X 0,Y 100.64,Z 382.949,A -85,B 0,C 180,E1 -26601.061,E2 -26601.061} C_VEL
LIN {X 0,Y 100.693,Z 382.936,A -85,B 0,C 180,E1 -26606.884,E2 -26606.884} C_VEL
LIN {X 0,Y 100.787,Z 382.924,A -85,B 0,C 180,E1 -26615.268,E2 -26615.268} C_VEL
LIN {X 0,Y 100.822,Z 382.925,A -85,B 0,C 180,E1 -26619.603,E2 -26619.603} C_VEL
LIN {X 0,Y 101.202,Z 382.879,A -85,B 0,C 180,E1 -26627.976,E2 -26627.976} C_VEL
LIN {X 0,Y 101.282,Z 382.861,A -85,B 0,C 180,E1 -26632.023,E2 -26632.023} C_VEL
LIN {X 0,Y 101.87,Z 382.788,A -85,B 0,C 180,E1 -26640.001,E2 -26640.001} C_VEL
LIN {X 0,Y 101.246,Z 382.867,A -85,B 0,C 180,E1 -26647.981,E2 -26647.981} C_VEL
LIN {X 0,Y 101.104,Z 382.891,A -85,B 0,C 180,E1 -26653.299,E2 -26653.299} C_VEL
LIN {X 0,Y 100.818,Z 382.927,A -85,B 0,C 180,E1 -26660.399,E2 -26660.399} C_VEL
LIN {X 0,Y 100.777,Z 382.925,A -85,B 0,C 180,E1 -26664.959,E2 -26664.959} C_VEL
LIN {X 0,Y 100.752,Z 382.93,A -85,B 0,C 180,E1 -26673.167,E2 -26673.167} C_VEL
LIN {X 0,Y 101.056,Z 382.896,A -85,B 0,C 180,E1 -26680.092,E2 -26680.092} C_VEL
LIN {X 0,Y 102.427,Z 382.729,A -85,B 0,C 180,E1 -26689.006,E2 -26689.006} C_VEL
LIN {X 0,Y 102.805,Z 382.89,A -85,B 0,C 180,E1 -26690.977,E2 -26690.977} C_VEL
LIN {X 0,Y 102.673,Z 385.033,A -85,B 0,C 180,E1 -26694.048,E2 -26694.048} C_VEL
LIN {X 0,Y 101.114,Z 391.934,A -85,B 0,C 180,E1 -26704.634,E2 -26704.634} C_VEL
LIN {X 0,Y 101.143,Z 394.104,A -85,B 0,C 180,E1 -26707.8,E2 -26707.8} C_VEL
LIN {X 0,Y 100.693,Z 407.047,A -85,B 0,C 180,E1 -26710.638,E2 -26710.638} C_VEL
LIN {X 0,Y 101.329,Z 420.784,A -85,B 0,C 180,E1 -26714.365,E2 -26714.365} C_VEL
LIN {X 0,Y 103.125,Z 434.011,A -85,B 0,C 180,E1 -26718.7,E2 -26718.7} C_VEL
LIN {X 0,Y 105.714,Z 445.868,A -85,B 0,C 180,E1 -26723.337,E2 -26723.337} C_VEL
LIN {X 0,Y 107.067,Z 451.051,A -85,B 0,C 180,E1 -26725.661,E2 -26725.661} C_VEL
LIN {X 0,Y 108.2,Z 458.511,A -85,B 0,C 180,E1 -26730,E2 -26730} C_VEL
LIN {X 0,Y 109.403,Z 463.919,A -85,B 0,C 180,E1 -26733.683,E2 -26733.683} C_VEL
LIN {X 0,Y 109.199,Z 465.75,A -85,B 0,C 180,E1 -26735.54,E2 -26735.54} C_VEL
LIN {X 0,Y 106.942,Z 470.451,A -85,B 0,C 180,E1 -26743.298,E2 -26743.298} C_VEL
LIN {X 0,Y 107.546,Z 474.808,A -85,B 0,C 180,E1 -26753.085,E2 -26753.085} C_VEL
LIN {X 0,Y 110.774,Z 477.301,A -85,B 0,C 180,E1 -26760.501,E2 -26760.501} C_VEL
LIN {X 0,Y 116.297,Z 479.094,A -85,B 0,C 180,E1 -26767.179,E2 -26767.179} C_VEL
LIN {X 0,Y 123.608,Z 480.158,A -85,B 0,C 180,E1 -26773.023,E2 -26773.023} C_VEL
LIN {X 0,Y 133.898,Z 480.421,A -85,B 0,C 180,E1 -26778.902,E2 -26778.902} C_VEL
LIN {X 0,Y 134.718,Z 479.906,A -85,B 0,C 180,E1 -26780.231,E2 -26780.231} C_VEL
LIN {X 0,Y 124.267,Z 474.226,A -85,B 0,C 180,E1 -26785.558,E2 -26785.558} C_VEL
LIN {X 0,Y 116.349,Z 467.943,A -85,B 0,C 180,E1 -26791.102,E2 -26791.102} C_VEL
LIN {X 0,Y 109.37,Z 459.364,A -85,B 0,C 180,E1 -26798.315,E2 -26798.315} C_VEL
LIN {X 0,Y 104.979,Z 450.106,A -85,B 0,C 180,E1 -26805.46,E2 -26805.46} C_VEL
LIN {X 0,Y 102.588,Z 439.103,A -85,B 0,C 180,E1 -26813.114,E2 -26813.114} C_VEL
LIN {X 0,Y 101.679,Z 427.346,A -85,B 0,C 180,E1 -26819.999,E2 -26819.999} C_VEL
LIN {X 0,Y 102.071,Z 415.309,A -85,B 0,C 180,E1 -26825.928,E2 -26825.928} C_VEL
LIN {X 0,Y 103.011,Z 401.827,A -85,B 0,C 180,E1 -26831.311,E2 -26831.311} C_VEL
LIN {X 0,Y 103.844,Z 391.399,A -85,B 0,C 180,E1 -26834.702,E2 -26834.702} C_VEL
LIN {X 0,Y 101.92,Z 382.78,A -85,B 0,C 180,E1 -26836.82,E2 -26836.82} C_VEL
LIN {X 0,Y 100.847,Z 382.916,A -85,B 0,C 180,E1 -26845.046,E2 -26845.046} C_VEL
LIN {X 0,Y 100.705,Z 382.935,A -85,B 0,C 180,E1 -26853.127,E2 -26853.127} C_VEL
LIN {X 0,Y 100.686,Z 382.935,A -85,B 0,C 180,E1 -26853.879,E2 -26853.879} C_VEL
LIN {X 0,Y 99.96,Z 383.033,A -85,B 0,C 180,E1 -26857.212,E2 -26857.212} C_VEL
LIN {X 0,Y 98.319,Z 383.236,A -85,B 0,C 180,E1 -26860.511,E2 -26860.511} C_VEL
LIN {X 0,Y 93.744,Z 383.804,A -85,B 0,C 180,E1 -26869.763,E2 -26869.763} C_VEL
LIN {X 0,Y 93.498,Z 383.829,A -85,B 0,C 180,E1 -26872.233,E2 -26872.233} C_VEL
LIN {X 0,Y 93.59,Z 383.823,A -85,B 0,C 180,E1 -26878.288,E2 -26878.288} C_VEL
LIN {X 0,Y 93.669,Z 383.818,A -85,B 0,C 180,E1 -26884.204,E2 -26884.204} C_VEL
LIN {X 0,Y 93.703,Z 383.806,A -85,B 0,C 180,E1 -26887.975,E2 -26887.975} C_VEL
LIN {X 0,Y 94.022,Z 383.766,A -85,B 0,C 180,E1 -26896.341,E2 -26896.341} C_VEL
LIN {X 0,Y 94.176,Z 383.754,A -85,B 0,C 180,E1 -26901.417,E2 -26901.417} C_VEL
LIN {X 0,Y 94.793,Z 383.678,A -85,B 0,C 180,E1 -26910,E2 -26910} C_VEL
LIN {X 0,Y 94.176,Z 383.754,A -85,B 0,C 180,E1 -26918.584,E2 -26918.584} C_VEL
LIN {X 0,Y 94.022,Z 383.766,A -85,B 0,C 180,E1 -26923.659,E2 -26923.659} C_VEL
LIN {X 0,Y 93.693,Z 383.807,A -85,B 0,C 180,E1 -26932.028,E2 -26932.028} C_VEL
LIN {X 0,Y 93.624,Z 383.822,A -85,B 0,C 180,E1 -26936.77,E2 -26936.77} C_VEL
LIN {X 0,Y 93.614,Z 383.824,A -85,B 0,C 180,E1 -26944.33,E2 -26944.33} C_VEL
LIN {X 0,Y 93.574,Z 383.829,A -85,B 0,C 180,E1 -26952.529,E2 -26952.529} C_VEL
LIN {X 0,Y 93.551,Z 383.827,A -85,B 0,C 180,E1 -26958.7,E2 -26958.7} C_VEL
LIN {X 0,Y 93.591,Z 383.819,A -85,B 0,C 180,E1 -26965.693,E2 -26965.693} C_VEL
LIN {X 0,Y 93.67,Z 383.809,A -85,B 0,C 180,E1 -26974.206,E2 -26974.206} C_VEL
LIN {X 0,Y 93.697,Z 383.813,A -85,B 0,C 180,E1 -26977.974,E2 -26977.974} C_VEL
LIN {X 0,Y 94.1,Z 383.764,A -85,B 0,C 180,E1 -26987.053,E2 -26987.053} C_VEL
LIN {X 0,Y 94.214,Z 383.741,A -85,B 0,C 180,E1 -26991.421,E2 -26991.421} C_VEL
LIN {X 0,Y 94.795,Z 383.669,A -85,B 0,C 180,E1 -27000.001,E2 -27000.001} C_VEL
LIN {X 0,Y 94.178,Z 383.746,A -85,B 0,C 180,E1 -27008.584,E2 -27008.584} C_VEL
LIN {X 0,Y 94.024,Z 383.773,A -85,B 0,C 180,E1 -27013.659,E2 -27013.659} C_VEL
LIN {X 0,Y 93.696,Z 383.814,A -85,B 0,C 180,E1 -27022.028,E2 -27022.028} C_VEL
LIN {X 0,Y 93.627,Z 383.817,A -85,B 0,C 180,E1 -27026.769,E2 -27026.769} C_VEL
LIN {X 0,Y 93.697,Z 383.806,A -85,B 0,C 180,E1 -27034.402,E2 -27034.402} C_VEL
LIN {X 0,Y 94.19,Z 383.748,A -85,B 0,C 180,E1 -27042.187,E2 -27042.187} C_VEL
LIN {X 0,Y 95.166,Z 383.633,A -85,B 0,C 180,E1 -27048.344,E2 -27048.344} C_VEL
LIN {X 0,Y 95.767,Z 383.554,A -85,B 0,C 180,E1 -27051.409,E2 -27051.409} C_VEL
LIN {X 0,Y 95.695,Z 383.681,A -85,B 0,C 180,E1 -27053.136,E2 -27053.136} C_VEL
LIN {X 0,Y 94.433,Z 388.513,A -85,B 0,C 180,E1 -27061.069,E2 -27061.069} C_VEL
LIN {X 0,Y 94.269,Z 392.91,A -85,B 0,C 180,E1 -27068.544,E2 -27068.544} C_VEL
LIN {X 0,Y 93.878,Z 405.182,A -85,B 0,C 180,E1 -27071.447,E2 -27071.447} C_VEL
LIN {X 0,Y 94.514,Z 418.114,A -85,B 0,C 180,E1 -27075.17,E2 -27075.17} C_VEL
LIN {X 0,Y 96.256,Z 430.713,A -85,B 0,C 180,E1 -27079.482,E2 -27079.482} C_VEL
LIN {X 0,Y 98.902,Z 442.502,A -85,B 0,C 180,E1 -27084.184,E2 -27084.184} C_VEL
LIN {X 0,Y 100.763,Z 448.695,A -85,B 0,C 180,E1 -27087.001,E2 -27087.001} C_VEL
LIN {X 0,Y 102.256,Z 456.824,A -85,B 0,C 180,E1 -27091.969,E2 -27091.969} C_VEL
LIN {X 0,Y 103.282,Z 460.938,A -85,B 0,C 180,E1 -27094.879,E2 -27094.879} C_VEL
LIN {X 0,Y 103.178,Z 461.904,A -85,B 0,C 180,E1 -27095.864,E2 -27095.864} C_VEL
LIN {X 0,Y 101.087,Z 466.384,A -85,B 0,C 180,E1 -27103.258,E2 -27103.258} C_VEL
LIN {X 0,Y 100.952,Z 469.772,A -85,B 0,C 180,E1 -27110.37,E2 -27110.37} C_VEL
LIN {X 0,Y 103.198,Z 472.929,A -85,B 0,C 180,E1 -27118.471,E2 -27118.471} C_VEL
LIN {X 0,Y 107.96,Z 475.323,A -85,B 0,C 180,E1 -27125.865,E2 -27125.865} C_VEL
LIN {X 0,Y 116.569,Z 477.297,A -85,B 0,C 180,E1 -27133.656,E2 -27133.656} C_VEL
LIN {X 0,Y 124.677,Z 478.048,A -85,B 0,C 180,E1 -27138.702,E2 -27138.702} C_VEL
LIN {X 0,Y 126.088,Z 477.995,A -85,B 0,C 180,E1 -27139.654,E2 -27139.654} C_VEL
LIN {X 0,Y 116.287,Z 471.876,A -85,B 0,C 180,E1 -27144.959,E2 -27144.959} C_VEL
LIN {X 0,Y 108.479,Z 464.874,A -85,B 0,C 180,E1 -27150.928,E2 -27150.928} C_VEL
LIN {X 0,Y 101.648,Z 455.334,A -85,B 0,C 180,E1 -27158.716,E2 -27158.716} C_VEL
LIN {X 0,Y 97.547,Z 445.184,A -85,B 0,C 180,E1 -27166.457,E2 -27166.457} C_VEL
LIN {X 0,Y 95.675,Z 434.645,A -85,B 0,C 180,E1 -27173.673,E2 -27173.673} C_VEL
LIN {X 0,Y 94.969,Z 423.884,A -85,B 0,C 180,E1 -27179.999,E2 -27179.999} C_VEL
LIN {X 0,Y 95.33,Z 412.291,A -85,B 0,C 180,E1 -27185.817,E2 -27185.817} C_VEL
LIN {X 0,Y 96.224,Z 399.442,A -85,B 0,C 180,E1 -27191.053,E2 -27191.053} C_VEL
LIN {X 0,Y 96.785,Z 392.017,A -85,B 0,C 180,E1 -27193.616,E2 -27193.616} C_VEL
LIN {X 0,Y 95.632,Z 386.166,A -85,B 0,C 180,E1 -27195.176,E2 -27195.176} C_VEL
LIN {X 0,Y 95.05,Z 383.638,A -85,B 0,C 180,E1 -27195.911,E2 -27195.911} C_VEL
LIN {X 0,Y 93.695,Z 383.807,A -85,B 0,C 180,E1 -27206.747,E2 -27206.747} C_VEL
LIN {X 0,Y 93.608,Z 383.817,A -85,B 0,C 180,E1 -27214.323,E2 -27214.323} C_VEL
LIN {X 0,Y 93.563,Z 383.823,A -85,B 0,C 180,E1 -27222.534,E2 -27222.534} C_VEL
LIN {X 0,Y 93.554,Z 383.83,A -85,B 0,C 180,E1 -27228.695,E2 -27228.695} C_VEL
LIN {X 0,Y 93.498,Z 383.829,A -85,B 0,C 180,E1 -27232.233,E2 -27232.233} C_VEL
LIN {X 0,Y 93.251,Z 383.87,A -85,B 0,C 180,E1 -27234.637,E2 -27234.637} C_VEL
LIN {X 0,Y 91.976,Z 384.041,A -85,B 0,C 180,E1 -27238.212,E2 -27238.212} C_VEL
LIN {X 0,Y 88.859,Z 384.434,A -85,B 0,C 180,E1 -27244.266,E2 -27244.266} C_VEL
LIN {X 0,Y 86.946,Z 384.659,A -85,B 0,C 180,E1 -27249.436,E2 -27249.436} C_VEL
LIN {X 0,Y 86.673,Z 384.68,A -85,B 0,C 180,E1 -27252.116,E2 -27252.116} C_VEL
LIN {X 0,Y 86.931,Z 384.65,A -85,B 0,C 180,E1 -27255.964,E2 -27255.964} C_VEL
LIN {X 0,Y 87.085,Z 384.637,A -85,B 0,C 180,E1 -27260.712,E2 -27260.712} C_VEL
LIN {X 0,Y 87.719,Z 384.559,A -85,B 0,C 180,E1 -27270,E2 -27270} C_VEL
LIN {X 0,Y 87.085,Z 384.637,A -85,B 0,C 180,E1 -27279.289,E2 -27279.289} C_VEL
LIN {X 0,Y 86.931,Z 384.65,A -85,B 0,C 180,E1 -27284.037,E2 -27284.037} C_VEL
LIN {X 0,Y 86.646,Z 384.691,A -85,B 0,C 180,E1 -27288.933,E2 -27288.933} C_VEL
LIN {X 0,Y 86.586,Z 384.699,A -85,B 0,C 180,E1 -27296.768,E2 -27296.768} C_VEL
LIN {X 0,Y 86.537,Z 384.704,A -85,B 0,C 180,E1 -27305.696,E2 -27305.696} C_VEL
LIN {X 0,Y 86.509,Z 384.71,A -85,B 0,C 180,E1 -27313.017,E2 -27313.017} C_VEL
LIN {X 0,Y 86.469,Z 384.711,A -85,B 0,C 180,E1 -27319.443,E2 -27319.443} C_VEL
LIN {X 0,Y 86.535,Z 384.698,A -85,B 0,C 180,E1 -27325.355,E2 -27325.355} C_VEL
LIN {X 0,Y 86.586,Z 384.693,A -85,B 0,C 180,E1 -27333.235,E2 -27333.235} C_VEL
LIN {X 0,Y 86.668,Z 384.685,A -85,B 0,C 180,E1 -27341.074,E2 -27341.074} C_VEL
LIN {X 0,Y 86.971,Z 384.65,A -85,B 0,C 180,E1 -27345.971,E2 -27345.971} C_VEL
LIN {X 0,Y 87.121,Z 384.625,A -85,B 0,C 180,E1 -27350.716,E2 -27350.716} C_VEL
LIN {X 0,Y 87.722,Z 384.55,A -85,B 0,C 180,E1 -27360.001,E2 -27360.001} C_VEL
LIN {X 0,Y 87.087,Z 384.63,A -85,B 0,C 180,E1 -27369.289,E2 -27369.289} C_VEL
LIN {X 0,Y 86.933,Z 384.656,A -85,B 0,C 180,E1 -27374.037,E2 -27374.037} C_VEL
LIN {X 0,Y 86.648,Z 384.688,A -85,B 0,C 180,E1 -27378.932,E2 -27378.932} C_VEL
LIN {X 0,Y 86.588,Z 384.693,A -85,B 0,C 180,E1 -27386.768,E2 -27386.768} C_VEL
LIN {X 0,Y 86.672,Z 384.683,A -85,B 0,C 180,E1 -27395.817,E2 -27395.817} C_VEL
LIN {X 0,Y 87.633,Z 384.572,A -85,B 0,C 180,E1 -27406.203,E2 -27406.203} C_VEL
LIN {X 0,Y 88.482,Z 384.462,A -85,B 0,C 180,E1 -27410.547,E2 -27410.547} C_VEL
LIN {X 0,Y 88.71,Z 384.434,A -85,B 0,C 180,E1 -27412.397,E2 -27412.397} C_VEL
LIN {X 0,Y 88.138,Z 384.558,A -85,B 0,C 180,E1 -27416.07,E2 -27416.07} C_VEL
LIN {X 0,Y 87.423,Z 391.76,A -85,B 0,C 180,E1 -27429.408,E2 -27429.408} C_VEL
LIN {X 0,Y 87.205,Z 406.306,A -85,B 0,C 180,E1 -27433.311,E2 -27433.311} C_VEL
LIN {X 0,Y 88.136,Z 418.844,A -85,B 0,C 180,E1 -27437.333,E2 -27437.333} C_VEL
LIN {X 0,Y 90.337,Z 431.544,A -85,B 0,C 180,E1 -27442.073,E2 -27442.073} C_VEL
LIN {X 0,Y 93.525,Z 443.523,A -85,B 0,C 180,E1 -27447.308,E2 -27447.308} C_VEL
LIN {X 0,Y 94.719,Z 446.963,A -85,B 0,C 180,E1 -27448.937,E2 -27448.937} C_VEL
LIN {X 0,Y 96.495,Z 455.053,A -85,B 0,C 180,E1 -27454.176,E2 -27454.176} C_VEL
LIN {X 0,Y 97.261,Z 457.824,A -85,B 0,C 180,E1 -27456.222,E2 -27456.222} C_VEL
LIN {X 0,Y 95.44,Z 461.872,A -85,B 0,C 180,E1 -27462.763,E2 -27462.763} C_VEL
LIN {X 0,Y 95.218,Z 466.156,A -85,B 0,C 180,E1 -27471.657,E2 -27471.657} C_VEL
LIN {X 0,Y 97.817,Z 469.599,A -85,B 0,C 180,E1 -27480.436,E2 -27480.436} C_VEL
LIN {X 0,Y 102.85,Z 472.186,A -85,B 0,C 180,E1 -27487.951,E2 -27487.951} C_VEL
LIN {X 0,Y 113.635,Z 474.73,A -85,B 0,C 180,E1 -27497.131,E2 -27497.131} C_VEL
LIN {X 0,Y 115.603,Z 474.981,A -85,B 0,C 180,E1 -27498.389,E2 -27498.389} C_VEL
LIN {X 0,Y 116.754,Z 474.967,A -85,B 0,C 180,E1 -27499.408,E2 -27499.408} C_VEL
LIN {X 0,Y 108.399,Z 468.966,A -85,B 0,C 180,E1 -27504.301,E2 -27504.301} C_VEL
LIN {X 0,Y 99.804,Z 460.104,A -85,B 0,C 180,E1 -27511.619,E2 -27511.619} C_VEL
LIN {X 0,Y 94.019,Z 450.719,A -85,B 0,C 180,E1 -27519.202,E2 -27519.202} C_VEL
LIN {X 0,Y 90.28,Z 439.546,A -85,B 0,C 180,E1 -27527.638,E2 -27527.638} C_VEL
LIN {X 0,Y 88.791,Z 429.675,A -85,B 0,C 180,E1 -27534.321,E2 -27534.321} C_VEL
LIN {X 0,Y 88.386,Z 416.902,A -85,B 0,C 180,E1 -27541.708,E2 -27541.708} C_VEL
LIN {X 0,Y 88.875,Z 405.064,A -85,B 0,C 180,E1 -27547.382,E2 -27547.382} C_VEL
LIN {X 0,Y 89.715,Z 393.762,A -85,B 0,C 180,E1 -27551.866,E2 -27551.866} C_VEL
LIN {X 0,Y 89.695,Z 390.226,A -85,B 0,C 180,E1 -27553.018,E2 -27553.018} C_VEL
LIN {X 0,Y 88.34,Z 384.482,A -85,B 0,C 180,E1 -27554.56,E2 -27554.56} C_VEL
LIN {X 0,Y 86.643,Z 384.686,A -85,B 0,C 180,E1 -27566.841,E2 -27566.841} C_VEL
LIN {X 0,Y 86.529,Z 384.701,A -85,B 0,C 180,E1 -27575.687,E2 -27575.687} C_VEL
LIN {X 0,Y 86.5,Z 384.702,A -85,B 0,C 180,E1 -27583.01,E2 -27583.01} C_VEL
LIN {X 0,Y 86.473,Z 384.71,A -85,B 0,C 180,E1 -27589.444,E2 -27589.444} C_VEL
LIN {X 0,Y 86.543,Z 384.705,A -85,B 0,C 180,E1 -27595.357,E2 -27595.357} C_VEL
LIN {X 0,Y 86.585,Z 384.699,A -85,B 0,C 180,E1 -27603.233,E2 -27603.233} C_VEL
LIN {X 0,Y 86.67,Z 384.688,A -85,B 0,C 180,E1 -27611.074,E2 -27611.074} C_VEL
LIN {X 0,Y 86.673,Z 384.68,A -85,B 0,C 180,E1 -27612.116,E2 -27612.116} C_VEL
LIN {X 0,Y 86.151,Z 384.747,A -85,B 0,C 180,E1 -27616.012,E2 -27616.012} C_VEL
LIN {X 0,Y 84.82,Z 384.918,A -85,B 0,C 180,E1 -27619.894,E2 -27619.894} C_VEL
LIN {X 0,Y 80.205,Z 385.481,A -85,B 0,C 180,E1 -27633.637,E2 -27633.637} C_VEL
LIN {X 0,Y 79.968,Z 385.522,A -85,B 0,C 180,E1 -27640.124,E2 -27640.124} C_VEL
LIN {X 0,Y 79.744,Z 385.549,A -85,B 0,C 180,E1 -27645.332,E2 -27645.332} C_VEL
LIN {X 0,Y 79.513,Z 385.573,A -85,B 0,C 180,E1 -27650.705,E2 -27650.705} C_VEL
LIN {X 0,Y 79.484,Z 385.581,A -85,B 0,C 180,E1 -27657.849,E2 -27657.849} C_VEL
LIN {X 0,Y 79.395,Z 385.592,A -85,B 0,C 180,E1 -27662.082,E2 -27662.082} C_VEL
LIN {X 0,Y 79.394,Z 385.587,A -85,B 0,C 180,E1 -27668.291,E2 -27668.291} C_VEL
LIN {X 0,Y 79.415,Z 385.589,A -85,B 0,C 180,E1 -27675.071,E2 -27675.071} C_VEL
LIN {X 0,Y 79.391,Z 385.595,A -85,B 0,C 180,E1 -27682.819,E2 -27682.819} C_VEL
LIN {X 0,Y 79.38,Z 385.594,A -85,B 0,C 180,E1 -27687.913,E2 -27687.913} C_VEL
LIN {X 0,Y 79.527,Z 385.57,A -85,B 0,C 180,E1 -27693.778,E2 -27693.778} C_VEL
LIN {X 0,Y 79.526,Z 385.578,A -85,B 0,C 180,E1 -27699.3,E2 -27699.3} C_VEL
LIN {X 0,Y 79.843,Z 385.538,A -85,B 0,C 180,E1 -27705.526,E2 -27705.526} C_VEL
LIN {X 0,Y 80.003,Z 385.514,A -85,B 0,C 180,E1 -27709.882,E2 -27709.882} C_VEL
LIN {X 0,Y 80.649,Z 385.431,A -85,B 0,C 180,E1 -27720.001,E2 -27720.001} C_VEL
LIN {X 0,Y 79.97,Z 385.518,A -85,B 0,C 180,E1 -27730.124,E2 -27730.124} C_VEL
LIN {X 0,Y 79.746,Z 385.547,A -85,B 0,C 180,E1 -27735.332,E2 -27735.332} C_VEL
LIN {X 0,Y 79.515,Z 385.58,A -85,B 0,C 180,E1 -27740.705,E2 -27740.705} C_VEL
LIN {X 0,Y 79.49,Z 385.58,A -85,B 0,C 180,E1 -27747.853,E2 -27747.853} C_VEL
LIN {X 0,Y 79.65,Z 385.562,A -85,B 0,C 180,E1 -27757.426,E2 -27757.426} C_VEL
LIN {X 0,Y 80.471,Z 385.463,A -85,B 0,C 180,E1 -27765.677,E2 -27765.677} C_VEL
LIN {X 0,Y 81.452,Z 385.336,A -85,B 0,C 180,E1 -27770.948,E2 -27770.948} C_VEL
LIN {X 0,Y 81.535,Z 385.327,A -85,B 0,C 180,E1 -27772.887,E2 -27772.887} C_VEL
LIN {X 0,Y 80.544,Z 385.545,A -85,B 0,C 180,E1 -27780.012,E2 -27780.012} C_VEL
LIN {X 0,Y 80.625,Z 390.676,A -85,B 0,C 180,E1 -27790.59,E2 -27790.59} C_VEL
LIN {X 0,Y 80.619,Z 405.784,A -85,B 0,C 180,E1 -27795.051,E2 -27795.051} C_VEL
LIN {X 0,Y 81.804,Z 418.388,A -85,B 0,C 180,E1 -27799.48,E2 -27799.48} C_VEL
LIN {X 0,Y 84.165,Z 430.278,A -85,B 0,C 180,E1 -27804.237,E2 -27804.237} C_VEL
LIN {X 0,Y 87.502,Z 441.598,A -85,B 0,C 180,E1 -27809.424,E2 -27809.424} C_VEL
LIN {X 0,Y 88.793,Z 445.068,A -85,B 0,C 180,E1 -27811.134,E2 -27811.134} C_VEL
LIN {X 0,Y 90.487,Z 451.725,A -85,B 0,C 180,E1 -27815.571,E2 -27815.571} C_VEL
LIN {X 0,Y 91.191,Z 454.443,A -85,B 0,C 180,E1 -27817.751,E2 -27817.751} C_VEL
LIN {X 0,Y 89.304,Z 460.262,A -85,B 0,C 180,E1 -27828.348,E2 -27828.348} C_VEL
LIN {X 0,Y 90.692,Z 464.265,A -85,B 0,C 180,E1 -27837.708,E2 -27837.708} C_VEL
LIN {X 0,Y 94.894,Z 467.492,A -85,B 0,C 180,E1 -27846.334,E2 -27846.334} C_VEL
LIN {X 0,Y 101.551,Z 470.032,A -85,B 0,C 180,E1 -27853.794,E2 -27853.794} C_VEL
LIN {X 0,Y 105.594,Z 471.029,A -85,B 0,C 180,E1 -27857.065,E2 -27857.065} C_VEL
LIN {X 0,Y 107.473,Z 471.107,A -85,B 0,C 180,E1 -27859.161,E2 -27859.161} C_VEL
LIN {X 0,Y 97.57,Z 462.419,A -85,B 0,C 180,E1 -27866.065,E2 -27866.065} C_VEL
LIN {X 0,Y 90.502,Z 453.3,A -85,B 0,C 180,E1 -27873.479,E2 -27873.479} C_VEL
LIN {X 0,Y 85.48,Z 442.543,A -85,B 0,C 180,E1 -27882.041,E2 -27882.041} C_VEL
LIN {X 0,Y 82.921,Z 431.448,A -85,B 0,C 180,E1 -27890.24,E2 -27890.24} C_VEL
LIN {X 0,Y 81.829,Z 419.011,A -85,B 0,C 180,E1 -27898.154,E2 -27898.154} C_VEL
LIN {X 0,Y 82.041,Z 406.362,A -85,B 0,C 180,E1 -27904.913,E2 -27904.913} C_VEL
LIN {X 0,Y 82.796,Z 393.726,A -85,B 0,C 180,E1 -27910.391,E2 -27910.391} C_VEL
LIN {X 0,Y 82.915,Z 390.386,A -85,B 0,C 180,E1 -27911.613,E2 -27911.613} C_VEL
LIN {X 0,Y 81.679,Z 385.312,A -85,B 0,C 180,E1 -27913.053,E2 -27913.053} C_VEL
LIN {X 0,Y 79.554,Z 385.573,A -85,B 0,C 180,E1 -27927.942,E2 -27927.942} C_VEL
LIN {X 0,Y 79.433,Z 385.588,A -85,B 0,C 180,E1 -27932.063,E2 -27932.063} C_VEL
LIN {X 0,Y 79.384,Z 385.596,A -85,B 0,C 180,E1 -27938.295,E2 -27938.295} C_VEL
LIN {X 0,Y 79.414,Z 385.59,A -85,B 0,C 180,E1 -27945.07,E2 -27945.07} C_VEL
LIN {X 0,Y 79.395,Z 385.589,A -85,B 0,C 180,E1 -27952.812,E2 -27952.812} C_VEL
LIN {X 0,Y 79.385,Z 385.593,A -85,B 0,C 180,E1 -27957.915,E2 -27957.915} C_VEL
LIN {X 0,Y 79.526,Z 385.579,A -85,B 0,C 180,E1 -27963.777,E2 -27963.777} C_VEL
LIN {X 0,Y 79.564,Z 385.559,A -85,B 0,C 180,E1 -27972.281,E2 -27972.281} C_VEL
LIN {X 0,Y 79.824,Z 385.536,A -85,B 0,C 180,E1 -27975.573,E2 -27975.573} C_VEL
LIN {X 0,Y 79.968,Z 385.522,A -85,B 0,C 180,E1 -27979.877,E2 -27979.877} C_VEL
LIN {X 0,Y 80.646,Z 385.44,A -85,B 0,C 180,E1 -27990,E2 -27990} C_VEL
LIN {X 0,Y 80.205,Z 385.481,A -85,B 0,C 180,E1 -27993.637,E2 -27993.637} C_VEL
LIN {X 0,Y 79.683,Z 385.556,A -85,B 0,C 180,E1 -27996.428,E2 -27996.428} C_VEL
LIN {X 0,Y 78.693,Z 385.683,A -85,B 0,C 180,E1 -27999.186,E2 -27999.186} C_VEL
LIN {X 0,Y 76.005,Z 386.013,A -85,B 0,C 180,E1 -28004.731,E2 -28004.731} C_VEL
LIN {X 0,Y 72.566,Z 386.443,A -85,B 0,C 180,E1 -28013.788,E2 -28013.788} C_VEL
LIN {X 0,Y 72.299,Z 386.46,A -85,B 0,C 180,E1 -28016.995,E2 -28016.995} C_VEL
LIN {X 0,Y 72.377,Z 386.462,A -85,B 0,C 180,E1 -28019.083,E2 -28019.083} C_VEL
LIN {X 0,Y 72.314,Z 386.476,A -85,B 0,C 180,E1 -28025.671,E2 -28025.671} C_VEL
LIN {X 0,Y 72.27,Z 386.483,A -85,B 0,C 180,E1 -28032.901,E2 -28032.901} C_VEL
LIN {X 0,Y 72.301,Z 386.479,A -85,B 0,C 180,E1 -28041.046,E2 -28041.046} C_VEL
LIN {X 0,Y 72.298,Z 386.473,A -85,B 0,C 180,E1 -28044.321,E2 -28044.321} C_VEL
LIN {X 0,Y 72.375,Z 386.469,A -85,B 0,C 180,E1 -28050.954,E2 -28050.954} C_VEL
LIN {X 0,Y 72.402,Z 386.465,A -85,B 0,C 180,E1 -28057.153,E2 -28057.153} C_VEL
LIN {X 0,Y 72.759,Z 386.418,A -85,B 0,C 180,E1 -28065.004,E2 -28065.004} C_VEL
LIN {X 0,Y 72.887,Z 386.403,A -85,B 0,C 180,E1 -28068.882,E2 -28068.882} C_VEL
LIN {X 0,Y 73.574,Z 386.311,A -85,B 0,C 180,E1 -28080.001,E2 -28080.001} C_VEL
LIN {X 0,Y 72.861,Z 386.407,A -85,B 0,C 180,E1 -28091.124,E2 -28091.124} C_VEL
LIN {X 0,Y 72.576,Z 386.435,A -85,B 0,C 180,E1 -28096.889,E2 -28096.889} C_VEL
LIN {X 0,Y 72.397,Z 386.466,A -85,B 0,C 180,E1 -28102.85,E2 -28102.85} C_VEL
LIN {X 0,Y 72.402,Z 386.466,A -85,B 0,C 180,E1 -28109.116,E2 -28109.116} C_VEL
LIN {X 0,Y 72.672,Z 386.433,A -85,B 0,C 180,E1 -28119.314,E2 -28119.314} C_VEL
LIN {X 0,Y 73.979,Z 386.269,A -85,B 0,C 180,E1 -28129.466,E2 -28129.466} C_VEL
LIN {X 0,Y 73.994,Z 386.265,A -85,B 0,C 180,E1 -28135.257,E2 -28135.257} C_VEL
LIN {X 0,Y 73.298,Z 386.564,A -85,B 0,C 180,E1 -28145.197,E2 -28145.197} C_VEL
LIN {X 0,Y 73.939,Z 389.619,A -85,B 0,C 180,E1 -28152.15,E2 -28152.15} C_VEL
LIN {X 0,Y 74.067,Z 403.896,A -85,B 0,C 180,E1 -28156.727,E2 -28156.727} C_VEL
LIN {X 0,Y 75.332,Z 416.015,A -85,B 0,C 180,E1 -28161.28,E2 -28161.28} C_VEL
LIN {X 0,Y 78.337,Z 429.516,A -85,B 0,C 180,E1 -28167.032,E2 -28167.032} C_VEL
LIN {X 0,Y 82.08,Z 440.7,A -85,B 0,C 180,E1 -28172.453,E2 -28172.453} C_VEL
LIN {X 0,Y 83.608,Z 444.878,A -85,B 0,C 180,E1 -28174.822,E2 -28174.822} C_VEL
LIN {X 0,Y 85.064,Z 449.728,A -85,B 0,C 180,E1 -28178.313,E2 -28178.313} C_VEL
LIN {X 0,Y 85.273,Z 450.98,A -85,B 0,C 180,E1 -28179.487,E2 -28179.487} C_VEL
LIN {X 0,Y 83.784,Z 456.201,A -85,B 0,C 180,E1 -28189.605,E2 -28189.605} C_VEL
LIN {X 0,Y 85.435,Z 460.419,A -85,B 0,C 180,E1 -28199.575,E2 -28199.575} C_VEL
LIN {X 0,Y 90.103,Z 463.892,A -85,B 0,C 180,E1 -28208.739,E2 -28208.739} C_VEL
LIN {X 0,Y 98.246,Z 466.961,A -85,B 0,C 180,E1 -28217.299,E2 -28217.299} C_VEL
LIN {X 0,Y 98.94,Z 466.862,A -85,B 0,C 180,E1 -28218.575,E2 -28218.575} C_VEL
LIN {X 0,Y 89.934,Z 458.071,A -85,B 0,C 180,E1 -28225.488,E2 -28225.488} C_VEL
LIN {X 0,Y 83.003,Z 448.038,A -85,B 0,C 180,E1 -28233.606,E2 -28233.606} C_VEL
LIN {X 0,Y 78.729,Z 437.84,A -85,B 0,C 180,E1 -28241.793,E2 -28241.793} C_VEL
LIN {X 0,Y 76.508,Z 427.695,A -85,B 0,C 180,E1 -28249.413,E2 -28249.413} C_VEL
LIN {X 0,Y 75.411,Z 415.605,A -85,B 0,C 180,E1 -28257.328,E2 -28257.328} C_VEL
LIN {X 0,Y 75.486,Z 403.569,A -85,B 0,C 180,E1 -28264.003,E2 -28264.003} C_VEL
LIN {X 0,Y 76.106,Z 391.915,A -85,B 0,C 180,E1 -28269.299,E2 -28269.299} C_VEL
LIN {X 0,Y 76.141,Z 390.242,A -85,B 0,C 180,E1 -28269.965,E2 -28269.965} C_VEL
LIN {X 0,Y 75.049,Z 386.137,A -85,B 0,C 180,E1 -28271.306,E2 -28271.306} C_VEL
LIN {X 0,Y 72.739,Z 386.423,A -85,B 0,C 180,E1 -28282.735,E2 -28282.735} C_VEL
LIN {X 0,Y 72.443,Z 386.461,A -85,B 0,C 180,E1 -28289.176,E2 -28289.176} C_VEL
LIN {X 0,Y 72.31,Z 386.478,A -85,B 0,C 180,E1 -28298.964,E2 -28298.964} C_VEL
LIN {X 0,Y 72.265,Z 386.484,A -85,B 0,C 180,E1 -28307.096,E2 -28307.096} C_VEL
LIN {X 0,Y 72.301,Z 386.477,A -85,B 0,C 180,E1 -28314.322,E2 -28314.322} C_VEL
LIN {X 0,Y 72.374,Z 386.462,A -85,B 0,C 180,E1 -28320.953,E2 -28320.953} C_VEL
LIN {X 0,Y 72.402,Z 386.46,A -85,B 0,C 180,E1 -28327.153,E2 -28327.153} C_VEL
LIN {X 0,Y 72.744,Z 386.42,A -85,B 0,C 180,E1 -28335.041,E2 -28335.041} C_VEL
LIN {X 0,Y 72.858,Z 386.404,A -85,B 0,C 180,E1 -28338.877,E2 -28338.877} C_VEL
LIN {X 0,Y 73.572,Z 386.321,A -85,B 0,C 180,E1 -28350,E2 -28350} C_VEL
LIN {X 0,Y 72.859,Z 386.404,A -85,B 0,C 180,E1 -28361.124,E2 -28361.124} C_VEL
LIN {X 0,Y 72.574,Z 386.445,A -85,B 0,C 180,E1 -28366.89,E2 -28366.89} C_VEL
LIN {X 0,Y 72.394,Z 386.461,A -85,B 0,C 180,E1 -28372.85,E2 -28372.85} C_VEL
LIN {X 0,Y 72.299,Z 386.46,A -85,B 0,C 180,E1 -28376.995,E2 -28376.995} C_VEL
LIN {X 0,Y 72.03,Z 386.504,A -85,B 0,C 180,E1 -28380.099,E2 -28380.099} C_VEL
LIN {X 0,Y 70.703,Z 386.678,A -85,B 0,C 180,E1 -28384.724,E2 -28384.724} C_VEL
LIN {X 0,Y 67.46,Z 387.082,A -85,B 0,C 180,E1 -28392.645,E2 -28392.645} C_VEL
LIN {X 0,Y 65.412,Z 387.334,A -85,B 0,C 180,E1 -28399.529,E2 -28399.529} C_VEL
LIN {X 0,Y 65.062,Z 387.359,A -85,B 0,C 180,E1 -28403.128,E2 -28403.128} C_VEL
LIN {X 0,Y 65.255,Z 387.357,A -85,B 0,C 180,E1 -28409.499,E2 -28409.499} C_VEL
LIN {X 0,Y 65.242,Z 387.349,A -85,B 0,C 180,E1 -28414.477,E2 -28414.477} C_VEL
LIN {X 0,Y 65.653,Z 387.301,A -85,B 0,C 180,E1 -28424.46,E2 -28424.46} C_VEL
LIN {X 0,Y 65.785,Z 387.29,A -85,B 0,C 180,E1 -28427.664,E2 -28427.664} C_VEL
LIN {X 0,Y 66.497,Z 387.193,A -85,B 0,C 180,E1 -28440.001,E2 -28440.001} C_VEL
LIN {X 0,Y 65.757,Z 387.294,A -85,B 0,C 180,E1 -28452.344,E2 -28452.344} C_VEL
LIN {X 0,Y 65.382,Z 387.335,A -85,B 0,C 180,E1 -28458.814,E2 -28458.814} C_VEL
LIN {X 0,Y 65.249,Z 387.348,A -85,B 0,C 180,E1 -28465.522,E2 -28465.522} C_VEL
LIN {X 0,Y 65.284,Z 387.347,A -85,B 0,C 180,E1 -28472.566,E2 -28472.566} C_VEL
LIN {X 0,Y 65.792,Z 387.284,A -85,B 0,C 180,E1 -28481.603,E2 -28481.603} C_VEL
LIN {X 0,Y 66.541,Z 387.198,A -85,B 0,C 180,E1 -28487.676,E2 -28487.676} C_VEL
LIN {X 0,Y 66.886,Z 387.148,A -85,B 0,C 180,E1 -28490.916,E2 -28490.916} C_VEL
LIN {X 0,Y 66.563,Z 387.192,A -85,B 0,C 180,E1 -28498.134,E2 -28498.134} C_VEL
LIN {X 0,Y 66.626,Z 387.312,A -85,B 0,C 180,E1 -28511.152,E2 -28511.152} C_VEL
LIN {X 0,Y 67.354,Z 388.568,A -85,B 0,C 180,E1 -28514.099,E2 -28514.099} C_VEL
LIN {X 0,Y 67.734,Z 402.888,A -85,B 0,C 180,E1 -28519.16,E2 -28519.16} C_VEL
LIN {X 0,Y 69.334,Z 415.205,A -85,B 0,C 180,E1 -28524.182,E2 -28524.182} C_VEL
LIN {X 0,Y 72.573,Z 428.016,A -85,B 0,C 180,E1 -28530,E2 -28530} C_VEL
LIN {X 0,Y 76.878,Z 439.539,A -85,B 0,C 180,E1 -28535.837,E2 -28535.837} C_VEL
LIN {X 0,Y 78.333,Z 443.138,A -85,B 0,C 180,E1 -28537.991,E2 -28537.991} C_VEL
LIN {X 0,Y 79.343,Z 446.117,A -85,B 0,C 180,E1 -28540.204,E2 -28540.204} C_VEL
LIN {X 0,Y 79.205,Z 447.839,A -85,B 0,C 180,E1 -28542.562,E2 -28542.562} C_VEL
LIN {X 0,Y 78.518,Z 452.819,A -85,B 0,C 180,E1 -28553.002,E2 -28553.002} C_VEL
LIN {X 0,Y 80.39,Z 456.399,A -85,B 0,C 180,E1 -28561.637,E2 -28561.637} C_VEL
LIN {X 0,Y 87.359,Z 460.966,A -85,B 0,C 180,E1 -28573.61,E2 -28573.61} C_VEL
LIN {X 0,Y 90.038,Z 462.032,A -85,B 0,C 180,E1 -28576.448,E2 -28576.448} C_VEL
LIN {X 0,Y 90.58,Z 461.874,A -85,B 0,C 180,E1 -28577.968,E2 -28577.968} C_VEL
LIN {X 0,Y 81.436,Z 451.781,A -85,B 0,C 180,E1 -28585.877,E2 -28585.877} C_VEL
LIN {X 0,Y 74.932,Z 440.586,A -85,B 0,C 180,E1 -28595.034,E2 -28595.034} C_VEL
LIN {X 0,Y 71.246,Z 429.148,A -85,B 0,C 180,E1 -28604.259,E2 -28604.259} C_VEL
LIN {X 0,Y 69.363,Z 417.358,A -85,B 0,C 180,E1 -28612.723,E2 -28612.723} C_VEL
LIN {X 0,Y 69.024,Z 404.506,A -85,B 0,C 180,E1 -28620.728,E2 -28620.728} C_VEL
LIN {X 0,Y 69.42,Z 391.499,A -85,B 0,C 180,E1 -28627.269,E2 -28627.269} C_VEL
LIN {X 0,Y 69.057,Z 388.41,A -85,B 0,C 180,E1 -28628.411,E2 -28628.411} C_VEL
LIN {X 0,Y 68.59,Z 386.937,A -85,B 0,C 180,E1 -28629.026,E2 -28629.026} C_VEL
LIN {X 0,Y 65.464,Z 387.321,A -85,B 0,C 180,E1 -28645.43,E2 -28645.43} C_VEL
LIN {X 0,Y 65.232,Z 387.354,A -85,B 0,C 180,E1 -28652.594,E2 -28652.594} C_VEL
LIN {X 0,Y 65.2,Z 387.359,A -85,B 0,C 180,E1 -28661.015,E2 -28661.015} C_VEL
LIN {X 0,Y 65.214,Z 387.356,A -85,B 0,C 180,E1 -28669.714,E2 -28669.714} C_VEL
LIN {X 0,Y 65.254,Z 387.348,A -85,B 0,C 180,E1 -28679.496,E2 -28679.496} C_VEL
LIN {X 0,Y 65.244,Z 387.358,A -85,B 0,C 180,E1 -28684.477,E2 -28684.477} C_VEL
LIN {X 0,Y 65.642,Z 387.306,A -85,B 0,C 180,E1 -28694.49,E2 -28694.49} C_VEL
LIN {X 0,Y 65.763,Z 387.284,A -85,B 0,C 180,E1 -28697.659,E2 -28697.659} C_VEL
LIN {X 0,Y 66.495,Z 387.203,A -85,B 0,C 180,E1 -28710,E2 -28710} C_VEL
LIN {X 0,Y 65.755,Z 387.285,A -85,B 0,C 180,E1 -28722.343,E2 -28722.343} C_VEL
LIN {X 0,Y 65.38,Z 387.339,A -85,B 0,C 180,E1 -28728.814,E2 -28728.814} C_VEL
LIN {X 0,Y 65.201,Z 387.355,A -85,B 0,C 180,E1 -28736.896,E2 -28736.896} C_VEL
LIN {X 0,Y 65.204,Z 387.361,A -85,B 0,C 180,E1 -28742.611,E2 -28742.611} C_VEL
LIN {X 0,Y 65.206,Z 387.36,A -85,B 0,C 180,E1 -28751.022,E2 -28751.022} C_VEL
LIN {X 0,Y 65.213,Z 387.359,A -85,B 0,C 180,E1 -28759.714,E2 -28759.714} C_VEL
LIN {X 0,Y 65.062,Z 387.359,A -85,B 0,C 180,E1 -28763.128,E2 -28763.128} C_VEL
LIN {X 0,Y 64.719,Z 387.415,A -85,B 0,C 180,E1 -28766.581,E2 -28766.581} C_VEL
LIN {X 0,Y 63.391,Z 387.591,A -85,B 0,C 180,E1 -28771.742,E2 -28771.742} C_VEL
LIN {X 0,Y 60.408,Z 387.957,A -85,B 0,C 180,E1 -28780.653,E2 -28780.653} C_VEL
LIN {X 0,Y 58.812,Z 388.158,A -85,B 0,C 180,E1 -28788.393,E2 -28788.393} C_VEL
LIN {X 0,Y 58.767,Z 388.154,A -85,B 0,C 180,E1 -28792.384,E2 -28792.384} C_VEL
LIN {X 0,Y 59.387,Z 388.078,A -85,B 0,C 180,E1 -28800.001,E2 -28800.001} C_VEL
LIN {X 0,Y 58.803,Z 388.154,A -85,B 0,C 180,E1 -28806.865,E2 -28806.865} C_VEL
LIN {X 0,Y 58.519,Z 388.187,A -85,B 0,C 180,E1 -28816.095,E2 -28816.095} C_VEL
LIN {X 0,Y 58.179,Z 388.237,A -85,B 0,C 180,E1 -28828.896,E2 -28828.896} C_VEL
LIN {X 0,Y 58.35,Z 388.215,A -85,B 0,C 180,E1 -28837.031,E2 -28837.031} C_VEL
LIN {X 0,Y 59.104,Z 388.122,A -85,B 0,C 180,E1 -28845.519,E2 -28845.519} C_VEL
LIN {X 0,Y 59.612,Z 388.058,A -85,B 0,C 180,E1 -28853.879,E2 -28853.879} C_VEL
LIN {X 0,Y 59.253,Z 388.097,A -85,B 0,C 180,E1 -28861.676,E2 -28861.676} C_VEL
LIN {X 0,Y 59.5,Z 388.073,A -85,B 0,C 180,E1 -28870.902,E2 -28870.902} C_VEL
LIN {X 0,Y 60.876,Z 387.893,A -85,B 0,C 180,E1 -28876.65,E2 -28876.65} C_VEL
LIN {X 0,Y 61.733,Z 403.001,A -85,B 0,C 180,E1 -28882.641,E2 -28882.641} C_VEL
LIN {X 0,Y 64.053,Z 416.178,A -85,B 0,C 180,E1 -28888.568,E2 -28888.568} C_VEL
LIN {X 0,Y 67.747,Z 428.318,A -85,B 0,C 180,E1 -28894.462,E2 -28894.462} C_VEL
LIN {X 0,Y 72.563,Z 439.386,A -85,B 0,C 180,E1 -28900.331,E2 -28900.331} C_VEL
LIN {X 0,Y 73.502,Z 441.618,A -85,B 0,C 180,E1 -28901.847,E2 -28901.847} C_VEL
LIN {X 0,Y 73.872,Z 443.208,A -85,B 0,C 180,E1 -28903.485,E2 -28903.485} C_VEL
LIN {X 0,Y 73.394,Z 448.464,A -85,B 0,C 180,E1 -28914.711,E2 -28914.711} C_VEL
LIN {X 0,Y 75.564,Z 452.193,A -85,B 0,C 180,E1 -28923.921,E2 -28923.921} C_VEL
LIN {X 0,Y 81.074,Z 456.033,A -85,B 0,C 180,E1 -28933.907,E2 -28933.907} C_VEL
LIN {X 0,Y 82.643,Z 456.39,A -85,B 0,C 180,E1 -28937.13,E2 -28937.13} C_VEL
LIN {X 0,Y 73.202,Z 444.568,A -85,B 0,C 180,E1 -28946.491,E2 -28946.491} C_VEL
LIN {X 0,Y 67.136,Z 432.033,A -85,B 0,C 180,E1 -28956.885,E2 -28956.885} C_VEL
LIN {X 0,Y 64.491,Z 421.98,A -85,B 0,C 180,E1 -28964.999,E2 -28964.999} C_VEL
LIN {X 0,Y 62.919,Z 408.899,A -85,B 0,C 180,E1 -28974.39,E2 -28974.39} C_VEL
LIN {X 0,Y 62.724,Z 396.906,A -85,B 0,C 180,E1 -28981.604,E2 -28981.604} C_VEL
LIN {X 0,Y 62.776,Z 388.937,A -85,B 0,C 180,E1 -28985.621,E2 -28985.621} C_VEL
LIN {X 0,Y 62.411,Z 387.709,A -85,B 0,C 180,E1 -28986.059,E2 -28986.059} C_VEL
LIN {X 0,Y 58.252,Z 388.228,A -85,B 0,C 180,E1 -29008.853,E2 -29008.853} C_VEL
LIN {X 0,Y 58.052,Z 388.252,A -85,B 0,C 180,E1 -29017.25,E2 -29017.25} C_VEL
LIN {X 0,Y 58.025,Z 388.257,A -85,B 0,C 180,E1 -29026.611,E2 -29026.611} C_VEL
LIN {X 0,Y 58.039,Z 388.248,A -85,B 0,C 180,E1 -29032.739,E2 -29032.739} C_VEL
LIN {X 0,Y 58.159,Z 388.236,A -85,B 0,C 180,E1 -29037.765,E2 -29037.765} C_VEL
LIN {X 0,Y 58.152,Z 388.233,A -85,B 0,C 180,E1 -29041.091,E2 -29041.091} C_VEL
LIN {X 0,Y 58.53,Z 388.193,A -85,B 0,C 180,E1 -29053.861,E2 -29053.861} C_VEL
LIN {X 0,Y 58.802,Z 388.158,A -85,B 0,C 180,E1 -29063.136,E2 -29063.136} C_VEL
LIN {X 0,Y 59.385,Z 388.088,A -85,B 0,C 180,E1 -29070,E2 -29070} C_VEL
LIN {X 0,Y 58.8,Z 388.158,A -85,B 0,C 180,E1 -29076.865,E2 -29076.865} C_VEL
LIN {X 0,Y 58.516,Z 388.195,A -85,B 0,C 180,E1 -29086.094,E2 -29086.094} C_VEL
LIN {X 0,Y 58.155,Z 388.233,A -85,B 0,C 180,E1 -29098.909,E2 -29098.909} C_VEL
LIN {X 0,Y 58.047,Z 388.247,A -85,B 0,C 180,E1 -29107.257,E2 -29107.257} C_VEL
LIN {X 0,Y 58.026,Z 388.248,A -85,B 0,C 180,E1 -29116.613,E2 -29116.613} C_VEL
LIN {X 0,Y 58.033,Z 388.253,A -85,B 0,C 180,E1 -29123.038,E2 -29123.038} C_VEL
LIN {X 0,Y 58.152,Z 388.24,A -85,B 0,C 180,E1 -29131.092,E2 -29131.092} C_VEL
LIN {X 0,Y 58.539,Z 388.185,A -85,B 0,C 180,E1 -29143.836,E2 -29143.836} C_VEL
LIN {X 0,Y 58.767,Z 388.154,A -85,B 0,C 180,E1 -29152.384,E2 -29152.384} C_VEL
LIN {X 0,Y 58.633,Z 388.189,A -85,B 0,C 180,E1 -29156.191,E2 -29156.191} C_VEL
LIN {X 0,Y 57.878,Z 388.299,A -85,B 0,C 180,E1 -29159.975,E2 -29159.975} C_VEL
LIN {X 0,Y 56.057,Z 388.542,A -85,B 0,C 180,E1 -29165.7,E2 -29165.7} C_VEL
LIN {X 0,Y 51,Z 389.118,A -85,B 0,C 180,E1 -29185.201,E2 -29185.201} C_VEL
LIN {X 0,Y 51.211,Z 389.096,A -85,B 0,C 180,E1 -29194.57,E2 -29194.57} C_VEL
LIN {X 0,Y 51.689,Z 389.038,A -85,B 0,C 180,E1 -29202.832,E2 -29202.832} C_VEL
LIN {X 0,Y 52.073,Z 389,A -85,B 0,C 180,E1 -29207.559,E2 -29207.559} C_VEL
LIN {X 0,Y 52.468,Z 388.946,A -85,B 0,C 180,E1 -29213.486,E2 -29213.486} C_VEL
LIN {X 0,Y 52.339,Z 388.964,A -85,B 0,C 180,E1 -29217.512,E2 -29217.512} C_VEL
LIN {X 0,Y 54.307,Z 388.717,A -85,B 0,C 180,E1 -29239.75,E2 -29239.75} C_VEL
LIN {X 0,Y 54.711,Z 388.849,A -85,B 0,C 180,E1 -29240.759,E2 -29240.759} C_VEL
LIN {X 0,Y 55.999,Z 402.576,A -85,B 0,C 180,E1 -29246.739,E2 -29246.739} C_VEL
LIN {X 0,Y 59.076,Z 416.34,A -85,B 0,C 180,E1 -29253.41,E2 -29253.41} C_VEL
LIN {X 0,Y 63.746,Z 429.028,A -85,B 0,C 180,E1 -29259.883,E2 -29259.883} C_VEL
LIN {X 0,Y 68.022,Z 437.689,A -85,B 0,C 180,E1 -29264.541,E2 -29264.541} C_VEL
LIN {X 0,Y 68.531,Z 438.774,A -85,B 0,C 180,E1 -29265.303,E2 -29265.303} C_VEL
LIN {X 0,Y 68.278,Z 442.99,A -85,B 0,C 180,E1 -29274.313,E2 -29274.313} C_VEL
LIN {X 0,Y 71.835,Z 448.594,A -85,B 0,C 180,E1 -29288.492,E2 -29288.492} C_VEL
LIN {X 0,Y 73.625,Z 449.892,A -85,B 0,C 180,E1 -29291.928,E2 -29291.928} C_VEL
LIN {X 0,Y 75.495,Z 450.834,A -85,B 0,C 180,E1 -29295.716,E2 -29295.716} C_VEL
LIN {X 0,Y 66.972,Z 439.428,A -85,B 0,C 180,E1 -29304.747,E2 -29304.747} C_VEL
LIN {X 0,Y 60.834,Z 426.049,A -85,B 0,C 180,E1 -29316.149,E2 -29316.149} C_VEL
LIN {X 0,Y 57.855,Z 413.789,A -85,B 0,C 180,E1 -29325.938,E2 -29325.938} C_VEL
LIN {X 0,Y 56.754,Z 401.67,A -85,B 0,C 180,E1 -29334.67,E2 -29334.67} C_VEL
LIN {X 0,Y 56.509,Z 388.824,A -85,B 0,C 180,E1 -29342.287,E2 -29342.287} C_VEL
LIN {X 0,Y 56.285,Z 388.473,A -85,B 0,C 180,E1 -29342.669,E2 -29342.669} C_VEL
LIN {X 0,Y 51.341,Z 389.082,A -85,B 0,C 180,E1 -29364.246,E2 -29364.246} C_VEL
LIN {X 0,Y 51.057,Z 389.115,A -85,B 0,C 180,E1 -29374.321,E2 -29374.321} C_VEL
LIN {X 0,Y 50.992,Z 389.133,A -85,B 0,C 180,E1 -29386.439,E2 -29386.439} C_VEL
LIN {X 0,Y 51.053,Z 389.125,A -85,B 0,C 180,E1 -29396.589,E2 -29396.589} C_VEL
LIN {X 0,Y 51.026,Z 389.127,A -85,B 0,C 180,E1 -29405.594,E2 -29405.594} C_VEL
LIN {X 0,Y 51.472,Z 389.072,A -85,B 0,C 180,E1 -29414.153,E2 -29414.153} C_VEL
LIN {X 0,Y 51.68,Z 389.047,A -85,B 0,C 180,E1 -29422.185,E2 -29422.185} C_VEL
LIN {X 0,Y 52.268,Z 388.975,A -85,B 0,C 180,E1 -29430.001,E2 -29430.001} C_VEL
LIN {X 0,Y 51.677,Z 389.047,A -85,B 0,C 180,E1 -29437.817,E2 -29437.817} C_VEL
LIN {X 0,Y 51.386,Z 389.084,A -85,B 0,C 180,E1 -29446.792,E2 -29446.792} C_VEL
LIN {X 0,Y 51.026,Z 389.127,A -85,B 0,C 180,E1 -29454.407,E2 -29454.407} C_VEL
LIN {X 0,Y 51.038,Z 389.128,A -85,B 0,C 180,E1 -29464.29,E2 -29464.29} C_VEL
LIN {X 0,Y 50.993,Z 389.124,A -85,B 0,C 180,E1 -29476.442,E2 -29476.442} C_VEL
LIN {X 0,Y 51.053,Z 389.117,A -85,B 0,C 180,E1 -29486.59,E2 -29486.59} C_VEL
LIN {X 0,Y 51.027,Z 389.121,A -85,B 0,C 180,E1 -29495.596,E2 -29495.596} C_VEL
LIN {X 0,Y 51.484,Z 389.064,A -85,B 0,C 180,E1 -29504.157,E2 -29504.157} C_VEL
LIN {X 0,Y 51.707,Z 389.033,A -85,B 0,C 180,E1 -29512.511,E2 -29512.511} C_VEL
LIN {X 0,Y 52.271,Z 388.964,A -85,B 0,C 180,E1 -29520.001,E2 -29520.001} C_VEL
LIN {X 0,Y 51.679,Z 389.039,A -85,B 0,C 180,E1 -29527.817,E2 -29527.817} C_VEL
LIN {X 0,Y 51.388,Z 389.074,A -85,B 0,C 180,E1 -29536.793,E2 -29536.793} C_VEL
LIN {X 0,Y 51,Z 389.118,A -85,B 0,C 180,E1 -29545.201,E2 -29545.201} C_VEL
LIN {X 0,Y 50.261,Z 389.22,A -85,B 0,C 180,E1 -29551.871,E2 -29551.871} C_VEL
LIN {X 0,Y 48.915,Z 389.392,A -85,B 0,C 180,E1 -29558.605,E2 -29558.605} C_VEL
LIN {X 0,Y 46.845,Z 389.651,A -85,B 0,C 180,E1 -29568.003,E2 -29568.003} C_VEL
LIN {X 0,Y 45.026,Z 389.864,A -85,B 0,C 180,E1 -29583.31,E2 -29583.31} C_VEL
LIN {X 0,Y 48.661,Z 389.415,A -85,B 0,C 180,E1 -29605.221,E2 -29605.221} C_VEL
LIN {X 0,Y 48.912,Z 389.505,A -85,B 0,C 180,E1 -29605.744,E2 -29605.744} C_VEL
LIN {X 0,Y 50.758,Z 402.384,A -85,B 0,C 180,E1 -29611.983,E2 -29611.983} C_VEL
LIN {X 0,Y 54.209,Z 415.076,A -85,B 0,C 180,E1 -29618.48,E2 -29618.48} C_VEL
LIN {X 0,Y 59.395,Z 427.538,A -85,B 0,C 180,E1 -29624.938,E2 -29624.938} C_VEL
LIN {X 0,Y 63.039,Z 434.405,A -85,B 0,C 180,E1 -29628.573,E2 -29628.573} C_VEL
LIN {X 0,Y 63.447,Z 435.33,A -85,B 0,C 180,E1 -29629.409,E2 -29629.409} C_VEL
LIN {X 0,Y 64.59,Z 440.833,A -85,B 0,C 180,E1 -29642.959,E2 -29642.959} C_VEL
LIN {X 0,Y 66.68,Z 443.247,A -85,B 0,C 180,E1 -29649.227,E2 -29649.227} C_VEL
LIN {X 0,Y 68.526,Z 444.531,A -85,B 0,C 180,E1 -29654.116,E2 -29654.116} C_VEL
LIN {X 0,Y 59.99,Z 432.106,A -85,B 0,C 180,E1 -29664.142,E2 -29664.142} C_VEL
LIN {X 0,Y 54.922,Z 420.231,A -85,B 0,C 180,E1 -29674.412,E2 -29674.412} C_VEL
LIN {X 0,Y 51.822,Z 406.993,A -85,B 0,C 180,E1 -29685.267,E2 -29685.267} C_VEL
LIN {X 0,Y 50.65,Z 394.983,A -85,B 0,C 180,E1 -29693.947,E2 -29693.947} C_VEL
LIN {X 0,Y 50.472,Z 389.192,A -85,B 0,C 180,E1 -29697.771,E2 -29697.771} C_VEL
LIN {X 0,Y 44.687,Z 389.912,A -85,B 0,C 180,E1 -29719.331,E2 -29719.331} C_VEL
LIN {X 0,Y 44.025,Z 389.998,A -85,B 0,C 180,E1 -29728.613,E2 -29728.613} C_VEL
LIN {X 0,Y 43.818,Z 390.024,A -85,B 0,C 180,E1 -29739.907,E2 -29739.907} C_VEL
LIN {X 0,Y 43.846,Z 390.016,A -85,B 0,C 180,E1 -29753.266,E2 -29753.266} C_VEL
LIN {X 0,Y 43.845,Z 390.015,A -85,B 0,C 180,E1 -29761.258,E2 -29761.258} C_VEL
LIN {X 0,Y 44.255,Z 389.972,A -85,B 0,C 180,E1 -29772.331,E2 -29772.331} C_VEL
LIN {X 0,Y 44.536,Z 389.937,A -85,B 0,C 180,E1 -29780.921,E2 -29780.921} C_VEL
LIN {X 0,Y 45.142,Z 389.862,A -85,B 0,C 180,E1 -29790.001,E2 -29790.001} C_VEL
LIN {X 0,Y 44.53,Z 389.938,A -85,B 0,C 180,E1 -29799.081,E2 -29799.081} C_VEL
LIN {X 0,Y 44.153,Z 389.982,A -85,B 0,C 180,E1 -29808.564,E2 -29808.564} C_VEL
LIN {X 0,Y 43.848,Z 390.014,A -85,B 0,C 180,E1 -29818.741,E2 -29818.741} C_VEL
LIN {X 0,Y 43.812,Z 390.019,A -85,B 0,C 180,E1 -29829.916,E2 -29829.916} C_VEL
LIN {X 0,Y 43.846,Z 390.018,A -85,B 0,C 180,E1 -29843.27,E2 -29843.27} C_VEL
LIN {X 0,Y 43.846,Z 390.021,A -85,B 0,C 180,E1 -29851.259,E2 -29851.259} C_VEL
LIN {X 0,Y 44.259,Z 389.962,A -85,B 0,C 180,E1 -29862.322,E2 -29862.322} C_VEL
LIN {X 0,Y 44.555,Z 389.925,A -85,B 0,C 180,E1 -29870.926,E2 -29870.926} C_VEL
LIN {X 0,Y 45.144,Z 389.852,A -85,B 0,C 180,E1 -29880.001,E2 -29880.001} C_VEL
LIN {X 0,Y 44.531,Z 389.928,A -85,B 0,C 180,E1 -29889.082,E2 -29889.082} C_VEL
LIN {X 0,Y 44.157,Z 389.976,A -85,B 0,C 180,E1 -29898.563,E2 -29898.563} C_VEL
LIN {X 0,Y 43.913,Z 390.012,A -85,B 0,C 180,E1 -29908.696,E2 -29908.696} C_VEL
LIN {X 0,Y 44.297,Z 389.966,A -85,B 0,C 180,E1 -29919.395,E2 -29919.395} C_VEL
LIN {X 0,Y 45.203,Z 389.845,A -85,B 0,C 180,E1 -29931.544,E2 -29931.544} C_VEL
LIN {X 0,Y 45.026,Z 389.864,A -85,B 0,C 180,E1 -29943.31,E2 -29943.31} C_VEL
LIN {X 0,Y 44.391,Z 389.949,A -85,B 0,C 180,E1 -29948.45,E2 -29948.45} C_VEL
LIN {X 0,Y 41.559,Z 390.301,A -85,B 0,C 180,E1 -29965.373,E2 -29965.373} C_VEL
LIN {X 0,Y 42.736,Z 390.158,A -85,B 0,C 180,E1 -29970.454,E2 -29970.454} C_VEL
LIN {X 0,Y 43.108,Z 390.111,A -85,B 0,C 180,E1 -29971.17,E2 -29971.17} C_VEL
LIN {X 0,Y 43.65,Z 390.042,A -85,B 0,C 180,E1 -29972.018,E2 -29972.018} C_VEL
LIN {X 0,Y 46.769,Z 404.554,A -85,B 0,C 180,E1 -29979.732,E2 -29979.732} C_VEL
LIN {X 0,Y 51.231,Z 416.926,A -85,B 0,C 180,E1 -29986.197,E2 -29986.197} C_VEL
LIN {X 0,Y 56.831,Z 428.093,A -85,B 0,C 180,E1 -29991.777,E2 -29991.777} C_VEL
LIN {X 0,Y 58.65,Z 431.173,A -85,B 0,C 180,E1 -29993.384,E2 -29993.384} C_VEL
LIN {X 0,Y 60.288,Z 436.012,A -85,B 0,C 180,E1 -30005.652,E2 -30005.652} C_VEL
LIN {X 0,Y 61.831,Z 437.516,A -85,B 0,C 180,E1 -30012.367,E2 -30012.367} C_VEL
LIN {X 0,Y 54.162,Z 425.713,A -85,B 0,C 180,E1 -30021.948,E2 -30021.948} C_VEL
LIN {X 0,Y 49.732,Z 415.441,A -85,B 0,C 180,E1 -30030.914,E2 -30030.914} C_VEL
LIN {X 0,Y 46.339,Z 401.945,A -85,B 0,C 180,E1 -30042.341,E2 -30042.341} C_VEL
LIN {X 0,Y 44.856,Z 389.884,A -85,B 0,C 180,E1 -30051.53,E2 -30051.53} C_VEL
LIN {X 0,Y 41.713,Z 390.28,A -85,B 0,C 180,E1 -30059.998,E2 -30059.998} C_VEL
LIN {X 0,Y 37.283,Z 390.84,A -85,B 0,C 180,E1 -30082.147,E2 -30082.147} C_VEL
LIN {X 0,Y 36.777,Z 390.894,A -85,B 0,C 180,E1 -30094.978,E2 -30094.978} C_VEL
LIN {X 0,Y 36.735,Z 390.904,A -85,B 0,C 180,E1 -30100.071,E2 -30100.071} C_VEL
LIN {X 0,Y 36.729,Z 390.901,A -85,B 0,C 180,E1 -30109.939,E2 -30109.939} C_VEL
LIN {X 0,Y 36.726,Z 390.909,A -85,B 0,C 180,E1 -30114.964,E2 -30114.964} C_VEL
LIN {X 0,Y 37.067,Z 390.863,A -85,B 0,C 180,E1 -30131.437,E2 -30131.437} C_VEL
LIN {X 0,Y 37.338,Z 390.827,A -85,B 0,C 180,E1 -30139.151,E2 -30139.151} C_VEL
LIN {X 0,Y 38,Z 390.752,A -85,B 0,C 180,E1 -30150.001,E2 -30150.001} C_VEL
LIN {X 0,Y 37.327,Z 390.828,A -85,B 0,C 180,E1 -30160.853,E2 -30160.853} C_VEL
LIN {X 0,Y 37.055,Z 390.865,A -85,B 0,C 180,E1 -30168.507,E2 -30168.507} C_VEL
LIN {X 0,Y 36.729,Z 390.908,A -85,B 0,C 180,E1 -30185.034,E2 -30185.034} C_VEL
LIN {X 0,Y 36.732,Z 390.901,A -85,B 0,C 180,E1 -30190.066,E2 -30190.066} C_VEL
LIN {X 0,Y 36.729,Z 390.905,A -85,B 0,C 180,E1 -30199.943,E2 -30199.943} C_VEL
LIN {X 0,Y 36.725,Z 390.901,A -85,B 0,C 180,E1 -30204.965,E2 -30204.965} C_VEL
LIN {X 0,Y 37.081,Z 390.857,A -85,B 0,C 180,E1 -30221.383,E2 -30221.383} C_VEL
LIN {X 0,Y 37.352,Z 390.826,A -85,B 0,C 180,E1 -30229.156,E2 -30229.156} C_VEL
LIN {X 0,Y 38.002,Z 390.741,A -85,B 0,C 180,E1 -30240.002,E2 -30240.002} C_VEL
LIN {X 0,Y 37.329,Z 390.829,A -85,B 0,C 180,E1 -30250.854,E2 -30250.854} C_VEL
LIN {X 0,Y 37.064,Z 390.859,A -85,B 0,C 180,E1 -30258.536,E2 -30258.536} C_VEL
LIN {X 0,Y 36.949,Z 390.872,A -85,B 0,C 180,E1 -30274.796,E2 -30274.796} C_VEL
LIN {X 0,Y 37.276,Z 390.834,A -85,B 0,C 180,E1 -30281.047,E2 -30281.047} C_VEL
LIN {X 0,Y 37.685,Z 390.788,A -85,B 0,C 180,E1 -30288.246,E2 -30288.246} C_VEL
LIN {X 0,Y 37.923,Z 390.761,A -85,B 0,C 180,E1 -30296.222,E2 -30296.222} C_VEL
LIN {X 0,Y 39.587,Z 390.549,A -85,B 0,C 180,E1 -30319.773,E2 -30319.773} C_VEL
LIN {X 0,Y 43.108,Z 390.111,A -85,B 0,C 180,E1 -30331.17,E2 -30331.17} C_VEL
LIN {X 0,Y 43.15,Z 390.358,A -85,B 0,C 180,E1 -30332.915,E2 -30332.915} C_VEL
LIN {X 0,Y 41.749,Z 391.902,A -85,B 0,C 180,E1 -30336.663,E2 -30336.663} C_VEL
LIN {X 0,Y 40.686,Z 395.137,A -85,B 0,C 180,E1 -30341.791,E2 -30341.791} C_VEL
LIN {X 0,Y 40.989,Z 399.858,A -85,B 0,C 180,E1 -30346.75,E2 -30346.75} C_VEL
LIN {X 0,Y 41.743,Z 403.514,A -85,B 0,C 180,E1 -30348.913,E2 -30348.913} C_VEL
LIN {X 0,Y 43.544,Z 407.665,A -85,B 0,C 180,E1 -30350.528,E2 -30350.528} C_VEL
LIN {X 0,Y 48.006,Z 415.836,A -85,B 0,C 180,E1 -30353.379,E2 -30353.379} C_VEL
LIN {X 0,Y 53.747,Z 426.178,A -85,B 0,C 180,E1 -30358.143,E2 -30358.143} C_VEL
LIN {X 0,Y 54.48,Z 427.409,A -85,B 0,C 180,E1 -30358.831,E2 -30358.831} C_VEL
LIN {X 0,Y 56.245,Z 430.926,A -85,B 0,C 180,E1 -30368.665,E2 -30368.665} C_VEL
LIN {X 0,Y 55.356,Z 429.671,A -85,B 0,C 180,E1 -30370.379,E2 -30370.379} C_VEL
LIN {X 0,Y 47.654,Z 416.656,A -85,B 0,C 180,E1 -30381.185,E2 -30381.185} C_VEL
LIN {X 0,Y 42.608,Z 402.948,A -85,B 0,C 180,E1 -30393.023,E2 -30393.023} C_VEL
LIN {X 0,Y 40.01,Z 390.489,A -85,B 0,C 180,E1 -30403.413,E2 -30403.413} C_VEL
LIN {X 0,Y 36.875,Z 390.88,A -85,B 0,C 180,E1 -30411.143,E2 -30411.143} C_VEL
LIN {X 0,Y 31.062,Z 391.528,A -85,B 0,C 180,E1 -30433.075,E2 -30433.075} C_VEL
LIN {X 0,Y 29.759,Z 391.648,A -85,B 0,C 180,E1 -30448.183,E2 -30448.183} C_VEL
LIN {X 0,Y 29.544,Z 391.668,A -85,B 0,C 180,E1 -30465.529,E2 -30465.529} C_VEL
LIN {X 0,Y 29.506,Z 391.672,A -85,B 0,C 180,E1 -30481.552,E2 -30481.552} C_VEL
LIN {X 0,Y 29.88,Z 391.636,A -85,B 0,C 180,E1 -30490.184,E2 -30490.184} C_VEL
LIN {X 0,Y 30.116,Z 391.613,A -85,B 0,C 180,E1 -30496.505,E2 -30496.505} C_VEL
LIN {X 0,Y 30.817,Z 391.551,A -85,B 0,C 180,E1 -30510.001,E2 -30510.001} C_VEL
LIN {X 0,Y 30.105,Z 391.614,A -85,B 0,C 180,E1 -30523.501,E2 -30523.501} C_VEL
LIN {X 0,Y 29.864,Z 391.637,A -85,B 0,C 180,E1 -30529.73,E2 -30529.73} C_VEL
LIN {X 0,Y 29.499,Z 391.671,A -85,B 0,C 180,E1 -30538.458,E2 -30538.458} C_VEL
LIN {X 0,Y 29.544,Z 391.667,A -85,B 0,C 180,E1 -30555.534,E2 -30555.534} C_VEL
LIN {X 0,Y 29.51,Z 391.672,A -85,B 0,C 180,E1 -30571.558,E2 -30571.558} C_VEL
LIN {X 0,Y 29.89,Z 391.636,A -85,B 0,C 180,E1 -30580.141,E2 -30580.141} C_VEL
LIN {X 0,Y 30.129,Z 391.615,A -85,B 0,C 180,E1 -30586.513,E2 -30586.513} C_VEL
LIN {X 0,Y 30.82,Z 391.546,A -85,B 0,C 180,E1 -30600.002,E2 -30600.002} C_VEL
LIN {X 0,Y 30.11,Z 391.617,A -85,B 0,C 180,E1 -30613.5,E2 -30613.5} C_VEL
LIN {X 0,Y 29.905,Z 391.635,A -85,B 0,C 180,E1 -30619.938,E2 -30619.938} C_VEL
LIN {X 0,Y 29.646,Z 391.659,A -85,B 0,C 180,E1 -30628.305,E2 -30628.305} C_VEL
LIN {X 0,Y 30.398,Z 391.59,A -85,B 0,C 180,E1 -30646.083,E2 -30646.083} C_VEL
LIN {X 0,Y 30.771,Z 391.554,A -85,B 0,C 180,E1 -30662.819,E2 -30662.819} C_VEL
LIN {X 0,Y 37.85,Z 390.767,A -85,B 0,C 180,E1 -30698.004,E2 -30698.004} C_VEL
LIN {X 0,Y 39.333,Z 390.715,A -85,B 0,C 180,E1 -30700.292,E2 -30700.292} C_VEL
LIN {X 0,Y 43.238,Z 404.609,A -85,B 0,C 180,E1 -30707.744,E2 -30707.744} C_VEL
LIN {X 0,Y 48.006,Z 415.836,A -85,B 0,C 180,E1 -30713.379,E2 -30713.379} C_VEL
LIN {X 0,Y 48.274,Z 416.823,A -85,B 0,C 180,E1 -30714.726,E2 -30714.726} C_VEL
LIN {X 0,Y 47.805,Z 417.203,A -85,B 0,C 180,E1 -30717.961,E2 -30717.961} C_VEL
LIN {X 0,Y 46.298,Z 415.949,A -85,B 0,C 180,E1 -30723.187,E2 -30723.187} C_VEL
LIN {X 0,Y 45.04,Z 414.221,A -85,B 0,C 180,E1 -30726.858,E2 -30726.858} C_VEL
LIN {X 0,Y 43.214,Z 411.154,A -85,B 0,C 180,E1 -30731.78,E2 -30731.78} C_VEL
LIN {X 0,Y 40.999,Z 406.018,A -85,B 0,C 180,E1 -30739.054,E2 -30739.054} C_VEL
LIN {X 0,Y 39.644,Z 402.159,A -85,B 0,C 180,E1 -30743.483,E2 -30743.483} C_VEL
LIN {X 0,Y 38.948,Z 400.085,A -85,B 0,C 180,E1 -30745.453,E2 -30745.453} C_VEL
LIN {X 0,Y 36.364,Z 390.946,A -85,B 0,C 180,E1 -30753.257,E2 -30753.257} C_VEL
LIN {X 0,Y 30.187,Z 391.609,A -85,B 0,C 180,E1 -30766.535,E2 -30766.535} C_VEL
LIN {X 0,Y 23.319,Z 392.049,A -85,B 0,C 180,E1 -30797.538,E2 -30797.538} C_VEL
LIN {X 0,Y 22.288,Z 392.082,A -85,B 0,C 180,E1 -30819.094,E2 -30819.094} C_VEL
LIN {X 0,Y 22.199,Z 392.085,A -85,B 0,C 180,E1 -30830.715,E2 -30830.715} C_VEL
LIN {X 0,Y 22.832,Z 392.065,A -85,B 0,C 180,E1 -30852.073,E2 -30852.073} C_VEL
LIN {X 0,Y 23.586,Z 392.041,A -85,B 0,C 180,E1 -30870.001,E2 -30870.001} C_VEL
LIN {X 0,Y 22.813,Z 392.065,A -85,B 0,C 180,E1 -30887.944,E2 -30887.944} C_VEL
LIN {X 0,Y 22.196,Z 392.084,A -85,B 0,C 180,E1 -30909.293,E2 -30909.293} C_VEL
LIN {X 0,Y 22.2,Z 392.084,A -85,B 0,C 180,E1 -30920.72,E2 -30920.72} C_VEL
LIN {X 0,Y 22.842,Z 392.064,A -85,B 0,C 180,E1 -30942.084,E2 -30942.084} C_VEL
LIN {X 0,Y 23.589,Z 392.042,A -85,B 0,C 180,E1 -30960.003,E2 -30960.003} C_VEL
LIN {X 0,Y 22.851,Z 392.064,A -85,B 0,C 180,E1 -30977.915,E2 -30977.915} C_VEL
LIN {X 0,Y 22.678,Z 392.069,A -85,B 0,C 180,E1 -30998.306,E2 -30998.306} C_VEL
LIN {X 0,Y 23.166,Z 392.054,A -85,B 0,C 180,E1 -31012.644,E2 -31012.644} C_VEL
LIN {X 0,Y 23.618,Z 392.04,A -85,B 0,C 180,E1 -31023.222,E2 -31023.222} C_VEL
LIN {X 0,Y 28.248,Z 391.789,A -85,B 0,C 180,E1 -31055.595,E2 -31055.595} C_VEL
LIN {X 0,Y 34.151,Z 391.228,A -85,B 0,C 180,E1 -31067.979,E2 -31067.979} C_VEL
LIN {X 0,Y 35.992,Z 391.029,A -85,B 0,C 180,E1 -31070.167,E2 -31070.167} C_VEL
LIN {X 0,Y 41.081,Z 405.188,A -85,B 0,C 180,E1 -31077.317,E2 -31077.317} C_VEL
LIN {X 0,Y 47.289,Z 417.508,A -85,B 0,C 180,E1 -31082.597,E2 -31082.597} C_VEL
LIN {X 0,Y 49.905,Z 421.817,A -85,B 0,C 180,E1 -31084.285,E2 -31084.285} C_VEL
LIN {X 0,Y 50.548,Z 422.937,A -85,B 0,C 180,E1 -31086.622,E2 -31086.622} C_VEL
LIN {X 0,Y 43.853,Z 411.814,A -85,B 0,C 180,E1 -31095.479,E2 -31095.479} C_VEL
LIN {X 0,Y 38.948,Z 400.085,A -85,B 0,C 180,E1 -31105.453,E2 -31105.453} C_VEL
LIN {X 0,Y 37.217,Z 397.313,A -85,B 0,C 180,E1 -31108.246,E2 -31108.246} C_VEL
LIN {X 0,Y 34.601,Z 395.244,A -85,B 0,C 180,E1 -31111.186,E2 -31111.186} C_VEL
LIN {X 0,Y 29.819,Z 393.273,A -85,B 0,C 180,E1 -31116.282,E2 -31116.282} C_VEL
LIN {X 0,Y 24.512,Z 392.406,A -85,B 0,C 180,E1 -31123.338,E2 -31123.338} C_VEL
LIN {X 0,Y 18.202,Z 392.178,A -85,B 0,C 180,E1 -31139.651,E2 -31139.651} C_VEL
LIN {X 0,Y 16.216,Z 392.178,A -85,B 0,C 180,E1 -31152.595,E2 -31152.595} C_VEL
LIN {X 0,Y 15.378,Z 392.178,A -85,B 0,C 180,E1 -31167.19,E2 -31167.19} C_VEL
LIN {X 0,Y 15.283,Z 392.178,A -85,B 0,C 180,E1 -31206.87,E2 -31206.87} C_VEL
LIN {X 0,Y 16.256,Z 392.178,A -85,B 0,C 180,E1 -31230.002,E2 -31230.002} C_VEL
LIN {X 0,Y 15.258,Z 392.178,A -85,B 0,C 180,E1 -31252.904,E2 -31252.904} C_VEL
LIN {X 0,Y 15.069,Z 392.178,A -85,B 0,C 180,E1 -31257.802,E2 -31257.802} C_VEL
LIN {X 0,Y 15.11,Z 392.178,A -85,B 0,C 180,E1 -31292.287,E2 -31292.287} C_VEL
LIN {X 0,Y 15.289,Z 392.178,A -85,B 0,C 180,E1 -31296.841,E2 -31296.841} C_VEL
LIN {X 0,Y 16.266,Z 392.178,A -85,B 0,C 180,E1 -31320.004,E2 -31320.004} C_VEL
LIN {X 0,Y 15.368,Z 392.178,A -85,B 0,C 180,E1 -31347.219,E2 -31347.219} C_VEL
LIN {X 0,Y 16.227,Z 392.178,A -85,B 0,C 180,E1 -31380.03,E2 -31380.03} C_VEL
LIN {X 0,Y 16.505,Z 392.178,A -85,B 0,C 180,E1 -31384.796,E2 -31384.796} C_VEL
LIN {X 0,Y 23.441,Z 392.046,A -85,B 0,C 180,E1 -31427.445,E2 -31427.445} C_VEL
LIN {X 0,Y 32.752,Z 391.364,A -85,B 0,C 180,E1 -31440.867,E2 -31440.867} C_VEL
LIN {X 0,Y 33.969,Z 391.244,A -85,B 0,C 180,E1 -31441.611,E2 -31441.611} C_VEL
LIN {X 0,Y 39.848,Z 404.825,A -85,B 0,C 180,E1 -31447.307,E2 -31447.307} C_VEL
LIN {X 0,Y 40.076,Z 405.389,A -85,B 0,C 180,E1 -31449.815,E2 -31449.815} C_VEL
LIN {X 0,Y 35.025,Z 393.712,A -85,B 0,C 180,E1 -31459.295,E2 -31459.295} C_VEL
LIN {X 0,Y 34.108,Z 391.236,A -85,B 0,C 180,E1 -31461.345,E2 -31461.345} C_VEL
LIN {X 0,Y 22.641,Z 392.07,A -85,B 0,C 180,E1 -31481.913,E2 -31481.913} C_VEL
LIN {X 0,Y 16.216,Z 392.178,A -85,B 0,C 180,E1 -31512.595,E2 -31512.595} C_VEL
LIN {X 0,Y 14.883,Z 392.178,A -85,B 0,C 180,E1 -31519.25,E2 -31519.25} C_VEL
LIN {X 0,Y 11.438,Z 392.178,A -85,B 0,C 180,E1 -31528.381,E2 -31528.381} C_VEL
LIN {X 0,Y 7.939,Z 392.178,A -85,B 0,C 180,E1 -31547.088,E2 -31547.088} C_VEL
LIN {X 0,Y 7.709,Z 392.178,A -85,B 0,C 180,E1 -31561.924,E2 -31561.924} C_VEL
LIN {X 0,Y 8.685,Z 392.178,A -85,B 0,C 180,E1 -31590.003,E2 -31590.003} C_VEL
LIN {X 0,Y 7.767,Z 392.178,A -85,B 0,C 180,E1 -31615.215,E2 -31615.215} C_VEL
LIN {X 0,Y 7.779,Z 392.178,A -85,B 0,C 180,E1 -31654.626,E2 -31654.626} C_VEL
LIN {X 0,Y 8.703,Z 392.178,A -85,B 0,C 180,E1 -31680.007,E2 -31680.007} C_VEL
LIN {X 0,Y 8.085,Z 392.178,A -85,B 0,C 180,E1 -31709.621,E2 -31709.621} C_VEL
LIN {X 0,Y 8.412,Z 392.178,A -85,B 0,C 180,E1 -31736.679,E2 -31736.679} C_VEL
LIN {X 0,Y 10.7,Z 392.178,A -85,B 0,C 180,E1 -31769.997,E2 -31769.997} C_VEL
LIN {X 0,Y 25.91,Z 391.969,A -85,B 0,C 180,E1 -31810.369,E2 -31810.369} C_VEL
LIN {X 0,Y 25.096,Z 391.994,A -85,B 0,C 180,E1 -31815.398,E2 -31815.398} C_VEL
LIN {X 0,Y 15.284,Z 392.178,A -85,B 0,C 180,E1 -31832.619,E2 -31832.619} C_VEL
LIN {X 0,Y 9.67,Z 392.178,A -85,B 0,C 180,E1 -31859.993,E2 -31859.993} C_VEL
LIN {X 0,Y 7.878,Z 392.178,A -85,B 0,C 180,E1 -31886.866,E2 -31886.866} C_VEL
LIN {X 0,Y 7.709,Z 392.178,A -85,B 0,C 180,E1 -31921.924,E2 -31921.924} C_VEL
LIN {X 0,Y 7.172,Z 392.178,A -85,B 0,C 180,E1 -31927.51,E2 -31927.51} C_VEL
LIN {X 0,Y 5.073,Z 392.178,A -85,B 0,C 180,E1 -31930.911,E2 -31930.911} C_VEL
LIN {X 0,Y 0.567,Z 392.178,A -85,B 0,C 180,E1 -31936.713,E2 -31936.713} C_VEL
LIN {X 0,Y 0.286,Z 392.178,A -85,B 0,C 180,E1 -32026.452,E2 -32026.452} C_VEL
LIN {X 0,Y 1.431,Z 392.178,A -85,B 0,C 180,E1 -32129.981,E2 -32129.981} C_VEL
LIN {X 0,Y 0.491,Z 392.178,A -85,B 0,C 180,E1 -32219.868,E2 -32219.868} C_VEL
LIN {X 0,Y 0.344,Z 392.178,A -85,B 0,C 180,E1 -32310.079,E2 -32310.079} C_VEL
LIN {X 0,Y 0.286,Z 392.178,A -85,B 0,C 180,E1 -32386.452,E2 -32386.452} C_VEL
LIN {X 0,Y 2.163,Z 394.178,A -85,B 0,C 180,E1 -32438.528,E2 -32438.528} C_VEL
LIN {X 0,Y 2.163,Z 600,A -85,B 0,C 180,E1 -32438.528,E2 -32438.528} C_VEL
LIN {X 0,Y 2.163,Z 600,A -85,B 0,C 180,E1 -32438.528,E2 -32438.528}

QRS_NEXT_CUT()

QRS_NEXT()
QRS_HOME()

END
